SPLINE
SPL {X  -159.063, Y  +688.696, Z    +0.000, E1   -17.094, E3 +447767.075}
SPL {X  -159.987, Y  +672.488, Z    +0.000, E1    -5.638, E3 +447791.140}
SPL {X  -159.990, Y  +663.928, Z    +0.000, E1    +0.338, E3 +447796.935}
SPL {X  -159.990, Y  +658.009, Z    +0.000, E1    +4.774, E3 +447800.634}
SPL {X  -159.990, Y  +651.567, Z    +0.000, E1    +9.674, E3 +447806.038}
SPL {X  -159.990, Y  +638.711, Z    +0.000, E1   +17.883, E3 +447821.684}
SPL {X  -159.990, Y  +631.642, Z    +0.000, E1   +20.884, E3 +447837.242}
SPL {X  -159.990, Y  +626.048, Z    +0.000, E1   +22.026, E3 +447857.236}
SPL {X  -159.990, Y  +623.760, Z    +0.000, E1   +22.031, E3 +447869.223}
SPL {X  -159.990, Y  +621.334, Z    +0.000, E1   +22.029, E3 +447881.949}
SPL {X  -159.990, Y  +618.387, Z    +0.000, E1   +22.057, E3 +447897.339}
SPL {X  -159.990, Y  +615.830, Z    +0.000, E1   +22.023, E3 +447910.830}
SPL {X  -159.990, Y  +613.034, Z    +0.000, E1   +22.053, E3 +447925.437}
SPL {X  -159.990, Y  +609.503, Z    +0.000, E1   +22.054, E3 +447943.964}
SPL {X  -159.990, Y  +605.804, Z    +0.000, E1   +22.064, E3 +447963.308}
SPL {X  -159.990, Y  +602.819, Z    +0.000, E1   +22.037, E3 +447978.979}
SPL {X  -159.990, Y  +600.642, Z    +0.000, E1   +22.032, E3 +447990.407}
SPL {X  -159.990, Y  +598.568, Z    +0.000, E1   +22.046, E3 +448001.200}
SPL {X  -159.990, Y  +596.440, Z    +0.000, E1   +22.036, E3 +448012.381}
SPL {X  -159.990, Y  +593.768, Z    +0.000, E1   +22.071, E3 +448026.314}
SPL {X  -159.990, Y  +590.068, Z    +0.000, E1   +22.076, E3 +448045.683}
SPL {X  -159.990, Y  +587.130, Z    +0.000, E1   +22.046, E3 +448061.120}
SPL {X  -159.990, Y  +585.120, Z    +0.000, E1   +22.045, E3 +448071.621}
SPL {X  -159.990, Y  +583.118, Z    +0.000, E1   +22.052, E3 +448082.108}
SPL {X  -159.990, Y  +580.862, Z    +0.000, E1   +22.049, E3 +448093.946}
SPL {X  -159.990, Y  +578.386, Z    +0.000, E1   +22.057, E3 +448106.901}
SPL {X  -159.990, Y  +576.252, Z    +0.000, E1   +22.038, E3 +448118.124}
SPL {X  -159.990, Y  +574.280, Z    +0.000, E1   +22.051, E3 +448128.418}
SPL {X  -159.990, Y  +571.711, Z    +0.000, E1   +22.058, E3 +448141.892}
SPL {X  -159.990, Y  +569.285, Z    +0.000, E1   +22.044, E3 +448154.617}
SPL {X  -159.990, Y  +567.211, Z    +0.000, E1   +22.046, E3 +448165.478}
SPL {X  -159.990, Y  +565.039, Z    +0.000, E1   +22.047, E3 +448176.856}
SPL {X  -159.990, Y  +562.755, Z    +0.000, E1   +22.047, E3 +448188.841}
SPL {X  -159.990, Y  +560.652, Z    +0.000, E1   +22.038, E3 +448199.886}
SPL {X  -159.990, Y  +558.852, Z    +0.000, E1   +22.046, E3 +448209.258}
SPL {X  -159.990, Y  +556.672, Z    +0.000, E1   +22.055, E3 +448220.647}
SPL {X  -159.990, Y  +553.726, Z    +0.000, E1   +22.080, E3 +448236.010}
SPL {X  -159.990, Y  +550.886, Z    +0.000, E1   +22.056, E3 +448250.948}
SPL {X  -159.990, Y  +548.814, Z    +0.000, E1   +22.049, E3 +448261.794}
SPL {X  -159.990, Y  +546.122, Z    +0.000, E1   +22.088, E3 +448275.808}
SPL {X  -159.990, Y  +542.390, Z    +0.000, E1   +22.086, E3 +448295.390}
SPL {X  -159.990, Y  +539.341, Z    +0.000, E1   +22.056, E3 +448311.411}
SPL {X  -159.990, Y  +536.301, Z    +0.000, E1   +22.084, E3 +448327.266}
SPL {X  -159.990, Y  +533.389, Z    +0.000, E1   +22.057, E3 +448342.573}
SPL {X  -159.990, Y  +531.347, Z    +0.000, E1   +22.052, E3 +448353.274}
SPL {X  -159.990, Y  +529.626, Z    +0.000, E1   +22.051, E3 +448362.271}
SPL {X  -159.990, Y  +527.412, Z    +0.000, E1   +22.067, E3 +448373.824}
SPL {X  -159.990, Y  +524.425, Z    +0.000, E1   +22.078, E3 +448389.456}
SPL {X  -159.990, Y  +521.599, Z    +0.000, E1   +22.060, E3 +448404.298}
SPL {X  -159.990, Y  +519.209, Z    +0.000, E1   +22.063, E3 +448416.773}
SPL {X  -159.990, Y  +517.330, Z    +0.000, E1   +22.053, E3 +448426.629}
SPL {X  -159.990, Y  +514.729, Z    +0.000, E1   +22.089, E3 +448440.187}
SPL {X  -159.990, Y  +511.670, Z    +0.000, E1   +22.064, E3 +448456.274}
SPL {X  -159.990, Y  +506.947, Z    +0.000, E1   +23.726, E3 +448466.303}
SPL {X  -159.990, Y  +496.921, Z    +0.000, E1   +28.340, E3 +448475.052}
SPL {X  -159.990, Y  +495.822, Z    +0.000, E1   +27.449, E3 +448485.800}
SPL {X  -159.990, Y  +494.952, Z    +0.000, E1   +26.628, E3 +448495.383}
SPL {X  -159.990, Y  +493.896, Z    +0.000, E1   +25.736, E3 +448506.713}
SPL {X  -159.990, Y  +491.647, Z    +0.000, E1   +25.401, E3 +448519.248}
SPL {X  -159.990, Y  +488.807, Z    +0.000, E1   +25.397, E3 +448531.947}
SPL {X  -159.990, Y  +486.070, Z    +0.000, E1   +25.399, E3 +448544.177}
SPL {X  -159.990, Y  +482.821, Z    +0.000, E1   +25.411, E3 +448558.679}
SPL {X  -159.990, Y  +480.183, Z    +0.000, E1   +25.384, E3 +448570.519}
SPL {X  -159.990, Y  +477.508, Z    +0.000, E1   +25.410, E3 +448582.428}
SPL {X  -159.990, Y  +473.634, Z    +0.000, E1   +25.426, E3 +448599.717}
SPL {X  -159.990, Y  +470.047, Z    +0.000, E1   +25.402, E3 +448615.798}
SPL {X  -159.990, Y  +466.213, Z    +0.000, E1   +25.433, E3 +448632.878}
SPL {X  -159.990, Y  +462.520, Z    +0.000, E1   +25.400, E3 +448649.446}
SPL {X  -159.990, Y  +460.081, Z    +0.000, E1   +25.390, E3 +448660.348}
SPL {X  -159.990, Y  +457.497, Z    +0.000, E1   +25.403, E3 +448671.872}
SPL {X  -159.990, Y  +455.126, Z    +0.000, E1   +25.389, E3 +448682.481}
SPL {X  -159.990, Y  +452.123, Z    +0.000, E1   +25.426, E3 +448695.838}
SPL {X  -159.990, Y  +448.503, Z    +0.000, E1   +25.410, E3 +448712.040}
SPL {X  -159.990, Y  +445.882, Z    +0.000, E1   +25.385, E3 +448723.842}
SPL {X  -159.990, Y  +443.345, Z    +0.000, E1   +25.390, E3 +448735.224}
SPL {X  -159.990, Y  +440.220, Z    +0.000, E1   +25.392, E3 +448749.212}
SPL {X  -159.990, Y  +436.316, Z    +0.000, E1   +25.420, E3 +448766.616}
SPL {X  -159.990, Y  +432.613, Z    +0.000, E1   +25.390, E3 +448783.241}
SPL {X  -159.990, Y  +429.079, Z    +0.000, E1   +25.407, E3 +448799.012}
SPL {X  -159.990, Y  +425.142, Z    +0.000, E1   +25.407, E3 +448816.614}
SPL {X  -159.990, Y  +421.010, Z    +0.000, E1   +25.418, E3 +448835.075}
SPL {X  -159.990, Y  +417.514, Z    +0.000, E1   +25.386, E3 +448850.768}
SPL {X  -159.990, Y  +414.805, Z    +0.000, E1   +25.385, E3 +448862.888}
SPL {X  -159.990, Y  +411.959, Z    +0.000, E1   +25.386, E3 +448875.615}
SPL {X  -159.990, Y  +408.981, Z    +0.000, E1   +25.392, E3 +448888.919}
SPL {X  -159.990, Y  +406.574, Z    +0.000, E1   +25.375, E3 +448899.693}
SPL {X  -159.990, Y  +403.513, Z    +0.000, E1   +25.420, E3 +448913.292}
SPL {X  -159.990, Y  +399.257, Z    +0.000, E1   +25.420, E3 +448932.333}
SPL {X  -159.990, Y  +395.992, Z    +0.000, E1   +25.380, E3 +448947.022}
SPL {X  -159.990, Y  +393.569, Z    +0.000, E1   +25.379, E3 +448957.866}
SPL {X  -159.990, Y  +390.564, Z    +0.000, E1   +25.393, E3 +448971.310}
SPL {X  -159.990, Y  +387.503, Z    +0.000, E1   +25.378, E3 +448985.024}
SPL {X  -159.990, Y  +384.900, Z    +0.000, E1   +25.383, E3 +448996.634}
SPL {X  -159.990, Y  +382.110, Z    +0.000, E1   +25.393, E3 +449009.080}
SPL {X  -159.961, Y  +379.439, Z    +0.000, E1   +25.380, E3 +449021.060}
SPL {X  -159.894, Y  +376.959, Z    +0.000, E1   +25.370, E3 +449032.237}
SPL {X  -159.784, Y  +374.382, Z    +0.000, E1   +25.356, E3 +449043.878}
SPL {X  -159.621, Y  +371.640, Z    +0.000, E1   +25.335, E3 +449056.318}
SPL {X  -159.406, Y  +368.844, Z    +0.000, E1   +25.307, E3 +449069.031}
SPL {X  -159.144, Y  +366.072, Z    +0.000, E1   +25.281, E3 +449081.638}
SPL {X  -158.822, Y  +363.200, Z    +0.000, E1   +25.236, E3 +449094.811}
SPL {X  -158.491, Y  +360.654, Z    +0.000, E1   +25.188, E3 +449106.551}
SPL {X  -158.127, Y  +358.155, Z    +0.000, E1   +25.126, E3 +449118.171}
SPL {X  -158.095, Y  +357.947, Z    +0.000, E1   +21.741, E3 +449149.743}
ENDSPLINE

SPLINE
SPL {X  -158.454, Y  +360.384, Z    +0.000, E1   +19.366, E3 +449161.894}
SPL {X  -159.737, Y  +373.507, Z    +0.000, E1   +10.311, E3 +449183.929}
SPL {X  -159.990, Y  +382.574, Z    +0.000, E1    +4.463, E3 +449190.617}
SPL {X  -159.990, Y  +389.909, Z    +0.000, E1    -0.662, E3 +449194.632}
SPL {X  -159.990, Y  +396.289, Z    +0.000, E1    -5.500, E3 +449198.412}
SPL {X  -159.990, Y  +407.941, Z    +0.000, E1   -14.126, E3 +449209.749}
SPL {X  -159.990, Y  +418.671, Z    +0.000, E1   -19.855, E3 +449229.165}
SPL {X  -159.990, Y  +429.878, Z    +0.000, E1   -23.330, E3 +449259.220}
SPL {X  -159.990, Y  +432.766, Z    +0.000, E1   -23.321, E3 +449273.443}
SPL {X  -159.990, Y  +434.794, Z    +0.000, E1   -23.304, E3 +449283.474}
SPL {X  -159.990, Y  +437.007, Z    +0.000, E1   -23.323, E3 +449294.326}
SPL {X  -159.990, Y  +439.778, Z    +0.000, E1   -23.323, E3 +449307.959}
SPL {X  -159.990, Y  +442.010, Z    +0.000, E1   -23.308, E3 +449318.980}
SPL {X  -159.990, Y  +443.729, Z    +0.000, E1   -23.310, E3 +449327.436}
SPL {X  -159.990, Y  +446.037, Z    +0.000, E1   -23.324, E3 +449338.773}
SPL {X  -159.990, Y  +449.434, Z    +0.000, E1   -23.356, E3 +449355.394}
SPL {X  -159.990, Y  +453.256, Z    +0.000, E1   -23.349, E3 +449374.229}
SPL {X  -159.990, Y  +455.953, Z    +0.000, E1   -23.320, E3 +449387.543}
SPL {X  -159.990, Y  +458.265, Z    +0.000, E1   -23.328, E3 +449398.898}
SPL {X  -159.990, Y  +461.258, Z    +0.000, E1   -23.344, E3 +449413.614}
SPL {X  -159.990, Y  +464.382, Z    +0.000, E1   -23.332, E3 +449428.995}
SPL {X  -159.990, Y  +466.881, Z    +0.000, E1   -23.322, E3 +449441.315}
SPL {X  -159.990, Y  +468.951, Z    +0.000, E1   -23.319, E3 +449451.507}
SPL {X  -159.990, Y  +471.818, Z    +0.000, E1   -23.351, E3 +449465.554}
SPL {X  -159.990, Y  +474.801, Z    +0.000, E1   -23.320, E3 +449480.330}
SPL {X  -159.990, Y  +476.830, Z    +0.000, E1   -23.323, E3 +449490.309}
SPL {X  -159.990, Y  +479.553, Z    +0.000, E1   -23.328, E3 +449503.711}
SPL {X  -159.990, Y  +482.950, Z    +0.000, E1   -23.350, E3 +449520.383}
SPL {X  -159.990, Y  +486.109, Z    +0.000, E1   -23.322, E3 +449535.999}
SPL {X  -159.990, Y  +489.247, Z    +0.000, E1   -23.348, E3 +449551.386}
SPL {X  -159.990, Y  +493.031, Z    +0.000, E1   -23.350, E3 +449570.010}
SPL {X  -159.990, Y  +496.869, Z    +0.000, E1   -23.349, E3 +449588.900}
SPL {X  -159.990, Y  +499.995, Z    +0.000, E1   -23.324, E3 +449604.334}
SPL {X  -159.990, Y  +502.456, Z    +0.000, E1   -23.324, E3 +449616.448}
SPL {X  -159.990, Y  +505.646, Z    +0.000, E1   -23.350, E3 +449632.103}
SPL {X  -159.990, Y  +508.862, Z    +0.000, E1   -23.328, E3 +449647.968}
SPL {X  -159.990, Y  +511.771, Z    +0.000, E1   -23.331, E3 +449662.290}
SPL {X  -159.990, Y  +514.016, Z    +0.000, E1   -23.308, E3 +449673.394}
SPL {X  -159.990, Y  +516.860, Z    +0.000, E1   -23.355, E3 +449687.280}
SPL {X  -159.990, Y  +520.719, Z    +0.000, E1   -23.363, E3 +449706.190}
SPL {X  -159.990, Y  +523.968, Z    +0.000, E1   -23.332, E3 +449722.275}
SPL {X  -159.990, Y  +526.466, Z    +0.000, E1   -23.320, E3 +449734.618}
SPL {X  -159.990, Y  +528.815, Z    +0.000, E1   -23.322, E3 +449746.178}
SPL {X  -159.990, Y  +531.246, Z    +0.000, E1   -23.325, E3 +449758.116}
SPL {X  -159.990, Y  +534.143, Z    +0.000, E1   -23.341, E3 +449772.351}
SPL {X  -159.990, Y  +537.024, Z    +0.000, E1   -23.321, E3 +449786.595}
SPL {X  -159.990, Y  +539.129, Z    +0.000, E1   -23.310, E3 +449796.978}
SPL {X  -159.990, Y  +541.882, Z    +0.000, E1   -23.346, E3 +449810.459}
SPL {X  -159.990, Y  +544.941, Z    +0.000, E1   -23.325, E3 +449825.541}
SPL {X  -159.990, Y  +548.126, Z    +0.000, E1   -23.354, E3 +449841.158}
SPL {X  -159.990, Y  +551.344, Z    +0.000, E1   -23.327, E3 +449857.050}
SPL {X  -159.990, Y  +553.642, Z    +0.000, E1   -23.319, E3 +449868.368}
SPL {X  -159.990, Y  +556.481, Z    +0.000, E1   -23.354, E3 +449882.275}
SPL {X  -159.990, Y  +559.475, Z    +0.000, E1   -23.321, E3 +449897.081}
SPL {X  -159.990, Y  +561.830, Z    +0.000, E1   -23.325, E3 +449908.666}
SPL {X  -159.990, Y  +564.273, Z    +0.000, E1   -23.325, E3 +449920.690}
SPL {X  -159.990, Y  +566.342, Z    +0.000, E1   -23.314, E3 +449930.894}
SPL {X  -159.990, Y  +568.849, Z    +0.000, E1   -23.338, E3 +449943.189}
SPL {X  -159.990, Y  +572.204, Z    +0.000, E1   -23.344, E3 +449959.684}
SPL {X  -159.990, Y  +575.097, Z    +0.000, E1   -23.325, E3 +449973.961}
SPL {X  -159.990, Y  +578.356, Z    +0.000, E1   -23.358, E3 +449989.933}
SPL {X  -159.990, Y  +582.292, Z    +0.000, E1   -23.360, E3 +450009.249}
SPL {X  -159.990, Y  +585.165, Z    +0.000, E1   -23.322, E3 +450023.492}
SPL {X  -159.990, Y  +587.388, Z    +0.000, E1   -23.328, E3 +450034.405}
SPL {X  -159.990, Y  +590.594, Z    +0.000, E1   -23.363, E3 +450050.097}
SPL {X  -159.990, Y  +594.301, Z    +0.000, E1   -23.358, E3 +450068.302}
SPL {X  -159.990, Y  +597.981, Z    +0.000, E1   -23.373, E3 +450086.350}
SPL {X  -159.990, Y  +600.935, Z    +0.000, E1   -23.343, E3 +450100.882}
SPL {X  -159.990, Y  +603.047, Z    +0.000, E1   -23.344, E3 +450111.268}
SPL {X  -159.990, Y  +605.187, Z    +0.000, E1   -23.344, E3 +450121.790}
SPL {X  -159.990, Y  +607.319, Z    +0.000, E1   -23.353, E3 +450132.252}
SPL {X  -159.990, Y  +610.569, Z    +0.000, E1   -23.372, E3 +450148.217}
SPL {X  -159.990, Y  +613.591, Z    +0.000, E1   -23.342, E3 +450163.145}
SPL {X  -159.990, Y  +615.604, Z    +0.000, E1   -23.330, E3 +450173.083}
SPL {X  -159.990, Y  +617.623, Z    +0.000, E1   -23.337, E3 +450183.014}
SPL {X  -159.990, Y  +620.788, Z    +0.000, E1   -23.368, E3 +450198.519}
SPL {X  -159.990, Y  +623.764, Z    +0.000, E1   -23.335, E3 +450213.211}
SPL {X  -159.990, Y  +626.608, Z    +0.000, E1   -23.361, E3 +450227.136}
SPL {X  -159.990, Y  +630.271, Z    +0.000, E1   -23.375, E3 +450245.097}
SPL {X  -159.990, Y  +633.318, Z    +0.000, E1   -23.339, E3 +450260.175}
SPL {X  -159.990, Y  +635.650, Z    +0.000, E1   -23.339, E3 +450271.646}
SPL {X  -159.990, Y  +637.839, Z    +0.000, E1   -23.335, E3 +450282.456}
SPL {X  -159.990, Y  +640.072, Z    +0.000, E1   -23.325, E3 +450293.488}
SPL {X  -159.990, Y  +642.230, Z    +0.000, E1   -23.323, E3 +450304.170}
SPL {X  -159.990, Y  +645.287, Z    +0.000, E1   -23.340, E3 +450319.196}
SPL {X  -159.990, Y  +648.792, Z    +0.000, E1   -23.346, E3 +450336.454}
SPL {X  -159.990, Y  +652.623, Z    +0.000, E1   -23.348, E3 +450355.289}
SPL {X  -159.990, Y  +656.380, Z    +0.000, E1   -23.347, E3 +450373.784}
SPL {X  -159.990, Y  +659.180, Z    +0.000, E1   -23.314, E3 +450387.632}
SPL {X  -159.990, Y  +661.392, Z    +0.000, E1   -23.318, E3 +450398.526}
SPL {X  -159.990, Y  +663.662, Z    +0.000, E1   -23.322, E3 +450409.650}
SPL {X  -159.990, Y  +665.964, Z    +0.000, E1   -23.328, E3 +450420.940}
SPL {X  -159.990, Y  +668.989, Z    +0.000, E1   -23.359, E3 +450435.776}
SPL {X  -159.990, Y  +671.893, Z    +0.000, E1   -23.319, E3 +450450.156}
SPL {X  -159.974, Y  +673.789, Z    +0.000, E1   -23.323, E3 +450459.472}
SPL {X  -159.924, Y  +676.110, Z    +0.000, E1   -23.320, E3 +450470.957}
SPL {X  -159.801, Y  +679.265, Z    +0.000, E1   -23.327, E3 +450486.575}
SPL {X  -159.626, Y  +682.287, Z    +0.000, E1   -23.280, E3 +450501.674}
SPL {X  -159.462, Y  +684.486, Z    +0.000, E1   -23.258, E3 +450512.673}
SPL {X  -159.246, Y  +686.911, Z    +0.000, E1   -23.230, E3 +450524.835}
SPL {X  -159.019, Y  +689.098, Z    +0.000, E1   -23.200, E3 +450535.837}
SPL {X  -158.660, Y  +692.086, Z    +0.000, E1   -23.176, E3 +450550.881}
ENDSPLINE

SPLINE
SPL {X  -159.063, Y  +688.696, Z    +0.000, E1   -17.094, E3 +450593.162}
SPL {X  -159.967, Y  +674.206, Z    +0.000, E1    -6.731, E3 +450615.975}
SPL {X  -159.990, Y  +665.270, Z    +0.000, E1    -0.699, E3 +450622.144}
SPL {X  -159.990, Y  +658.009, Z    +0.000, E1    +4.774, E3 +450626.721}
SPL {X  -159.990, Y  +651.567, Z    +0.000, E1    +9.674, E3 +450632.125}
SPL {X  -159.990, Y  +637.762, Z    +0.000, E1   +18.345, E3 +450649.483}
SPL {X  -159.990, Y  +626.382, Z    +0.000, E1   +22.040, E3 +450681.532}
SPL {X  -159.990, Y  +623.760, Z    +0.000, E1   +22.031, E3 +450695.310}
SPL {X  -159.990, Y  +621.334, Z    +0.000, E1   +22.029, E3 +450708.036}
SPL {X  -159.990, Y  +618.387, Z    +0.000, E1   +22.057, E3 +450723.426}
SPL {X  -159.990, Y  +614.928, Z    +0.000, E1   +22.055, E3 +450741.579}
SPL {X  -159.990, Y  +611.459, Z    +0.000, E1   +22.053, E3 +450759.782}
SPL {X  -159.990, Y  +608.810, Z    +0.000, E1   +22.023, E3 +450773.750}
SPL {X  -159.990, Y  +606.481, Z    +0.000, E1   +22.033, E3 +450785.925}
SPL {X  -159.990, Y  +603.419, Z    +0.000, E1   +22.064, E3 +450801.865}
SPL {X  -159.990, Y  +600.642, Z    +0.000, E1   +22.032, E3 +450816.494}
SPL {X  -159.990, Y  +598.568, Z    +0.000, E1   +22.046, E3 +450827.287}
SPL {X  -159.990, Y  +595.493, Z    +0.000, E1   +22.070, E3 +450843.370}
SPL {X  -159.990, Y  +592.865, Z    +0.000, E1   +22.036, E3 +450857.199}
SPL {X  -159.990, Y  +590.803, Z    +0.000, E1   +22.046, E3 +450867.989}
SPL {X  -159.990, Y  +587.778, Z    +0.000, E1   +22.073, E3 +450883.764}
SPL {X  -159.990, Y  +585.120, Z    +0.000, E1   +22.045, E3 +450897.708}
SPL {X  -159.990, Y  +583.118, Z    +0.000, E1   +22.052, E3 +450908.195}
SPL {X  -159.990, Y  +580.131, Z    +0.000, E1   +22.078, E3 +450923.801}
SPL {X  -159.990, Y  +576.888, Z    +0.000, E1   +22.061, E3 +450940.831}
SPL {X  -159.990, Y  +574.280, Z    +0.000, E1   +22.051, E3 +450954.505}
SPL {X  -159.990, Y  +571.711, Z    +0.000, E1   +22.058, E3 +450967.979}
SPL {X  -159.990, Y  +569.285, Z    +0.000, E1   +22.044, E3 +450980.704}
SPL {X  -159.990, Y  +567.211, Z    +0.000, E1   +22.046, E3 +450991.565}
SPL {X  -159.990, Y  +565.039, Z    +0.000, E1   +22.047, E3 +451002.942}
SPL {X  -159.990, Y  +562.755, Z    +0.000, E1   +22.047, E3 +451014.928}
SPL {X  -159.990, Y  +560.652, Z    +0.000, E1   +22.038, E3 +451025.973}
SPL {X  -159.990, Y  +558.852, Z    +0.000, E1   +22.046, E3 +451035.345}
SPL {X  -159.990, Y  +556.672, Z    +0.000, E1   +22.055, E3 +451046.734}
SPL {X  -159.990, Y  +553.726, Z    +0.000, E1   +22.080, E3 +451062.097}
SPL {X  -159.990, Y  +550.886, Z    +0.000, E1   +22.056, E3 +451077.035}
SPL {X  -159.990, Y  +548.814, Z    +0.000, E1   +22.049, E3 +451087.881}
SPL {X  -159.990, Y  +546.122, Z    +0.000, E1   +22.088, E3 +451101.895}
SPL {X  -159.990, Y  +542.390, Z    +0.000, E1   +22.086, E3 +451121.477}
SPL {X  -159.990, Y  +539.341, Z    +0.000, E1   +22.056, E3 +451137.498}
SPL {X  -159.990, Y  +536.984, Z    +0.000, E1   +22.057, E3 +451149.829}
SPL {X  -159.990, Y  +534.045, Z    +0.000, E1   +22.087, E3 +451165.154}
SPL {X  -159.990, Y  +530.476, Z    +0.000, E1   +22.084, E3 +451183.847}
SPL {X  -159.990, Y  +527.412, Z    +0.000, E1   +22.067, E3 +451199.911}
SPL {X  -159.990, Y  +524.425, Z    +0.000, E1   +22.078, E3 +451215.543}
SPL {X  -159.990, Y  +521.599, Z    +0.000, E1   +22.060, E3 +451230.385}
SPL {X  -159.990, Y  +519.209, Z    +0.000, E1   +22.063, E3 +451242.860}
SPL {X  -159.990, Y  +516.651, Z    +0.000, E1   +22.071, E3 +451256.239}
SPL {X  -159.990, Y  +514.122, Z    +0.000, E1   +22.061, E3 +451269.512}
SPL {X  -159.990, Y  +511.670, Z    +0.000, E1   +22.064, E3 +451282.361}
SPL {X  -159.990, Y  +506.947, Z    +0.000, E1   +23.726, E3 +451292.390}
SPL {X  -159.990, Y  +496.921, Z    +0.000, E1   +28.340, E3 +451301.139}
SPL {X  -159.990, Y  +495.822, Z    +0.000, E1   +27.449, E3 +451311.887}
SPL {X  -159.990, Y  +494.952, Z    +0.000, E1   +26.628, E3 +451321.470}
SPL {X  -159.990, Y  +493.896, Z    +0.000, E1   +25.736, E3 +451332.800}
SPL {X  -159.990, Y  +491.647, Z    +0.000, E1   +25.401, E3 +451345.335}
SPL {X  -159.990, Y  +488.807, Z    +0.000, E1   +25.397, E3 +451358.033}
SPL {X  -159.990, Y  +486.070, Z    +0.000, E1   +25.399, E3 +451370.264}
SPL {X  -159.990, Y  +483.747, Z    +0.000, E1   +25.384, E3 +451380.677}
SPL {X  -159.990, Y  +481.038, Z    +0.000, E1   +25.412, E3 +451392.733}
SPL {X  -159.990, Y  +477.508, Z    +0.000, E1   +25.410, E3 +451408.515}
SPL {X  -159.990, Y  +473.634, Z    +0.000, E1   +25.426, E3 +451425.804}
SPL {X  -159.990, Y  +470.047, Z    +0.000, E1   +25.402, E3 +451441.885}
SPL {X  -159.990, Y  +467.082, Z    +0.000, E1   +25.399, E3 +451455.132}
SPL {X  -159.990, Y  +464.063, Z    +0.000, E1   +25.405, E3 +451468.627}
SPL {X  -159.990, Y  +460.712, Z    +0.000, E1   +25.411, E3 +451483.587}
SPL {X  -159.990, Y  +457.497, Z    +0.000, E1   +25.403, E3 +451497.959}
SPL {X  -159.990, Y  +454.323, Z    +0.000, E1   +25.412, E3 +451512.118}
SPL {X  -159.990, Y  +450.823, Z    +0.000, E1   +25.417, E3 +451527.747}
SPL {X  -159.990, Y  +447.982, Z    +0.000, E1   +25.393, E3 +451540.488}
SPL {X  -159.990, Y  +445.108, Z    +0.000, E1   +25.407, E3 +451553.365}
SPL {X  -159.990, Y  +441.797, Z    +0.000, E1   +25.390, E3 +451568.244}
SPL {X  -159.990, Y  +439.442, Z    +0.000, E1   +25.369, E3 +451578.821}
SPL {X  -159.990, Y  +436.316, Z    +0.000, E1   +25.420, E3 +451592.703}
SPL {X  -159.990, Y  +432.613, Z    +0.000, E1   +25.390, E3 +451609.328}
SPL {X  -159.990, Y  +429.827, Z    +0.000, E1   +25.380, E3 +451621.805}
SPL {X  -159.990, Y  +426.865, Z    +0.000, E1   +25.398, E3 +451635.010}
SPL {X  -159.990, Y  +423.417, Z    +0.000, E1   +25.400, E3 +451650.426}
SPL {X  -159.990, Y  +420.283, Z    +0.000, E1   +25.386, E3 +451664.470}
SPL {X  -159.990, Y  +417.514, Z    +0.000, E1   +25.386, E3 +451676.855}
SPL {X  -159.990, Y  +414.805, Z    +0.000, E1   +25.385, E3 +451688.975}
SPL {X  -159.990, Y  +411.959, Z    +0.000, E1   +25.386, E3 +451701.702}
SPL {X  -159.990, Y  +408.981, Z    +0.000, E1   +25.392, E3 +451715.006}
SPL {X  -159.990, Y  +405.773, Z    +0.000, E1   +25.398, E3 +451729.315}
SPL {X  -159.990, Y  +402.805, Z    +0.000, E1   +25.389, E3 +451742.602}
SPL {X  -159.990, Y  +399.257, Z    +0.000, E1   +25.420, E3 +451758.420}
SPL {X  -159.990, Y  +395.992, Z    +0.000, E1   +25.380, E3 +451773.109}
SPL {X  -159.990, Y  +393.569, Z    +0.000, E1   +25.379, E3 +451783.952}
SPL {X  -159.990, Y  +390.564, Z    +0.000, E1   +25.393, E3 +451797.397}
SPL {X  -159.990, Y  +387.503, Z    +0.000, E1   +25.378, E3 +451811.111}
SPL {X  -159.990, Y  +384.900, Z    +0.000, E1   +25.383, E3 +451822.721}
SPL {X  -159.990, Y  +382.110, Z    +0.000, E1   +25.393, E3 +451835.167}
SPL {X  -159.961, Y  +379.439, Z    +0.000, E1   +25.380, E3 +451847.147}
SPL {X  -159.894, Y  +376.959, Z    +0.000, E1   +25.370, E3 +451858.324}
SPL {X  -159.784, Y  +374.382, Z    +0.000, E1   +25.356, E3 +451869.965}
SPL {X  -159.621, Y  +371.640, Z    +0.000, E1   +25.335, E3 +451882.405}
SPL {X  -159.406, Y  +368.844, Z    +0.000, E1   +25.307, E3 +451895.118}
SPL {X  -159.144, Y  +366.072, Z    +0.000, E1   +25.281, E3 +451907.725}
SPL {X  -158.822, Y  +363.200, Z    +0.000, E1   +25.236, E3 +451920.898}
SPL {X  -158.491, Y  +360.654, Z    +0.000, E1   +25.188, E3 +451932.638}
SPL {X  -158.127, Y  +358.155, Z    +0.000, E1   +25.126, E3 +451944.258}
SPL {X  -158.095, Y  +357.947, Z    +0.000, E1   +21.741, E3 +451975.830}
ENDSPLINE

SPLINE
SPL {X  -158.454, Y  +360.384, Z    +0.000, E1   +19.366, E3 +451987.981}
SPL {X  -159.737, Y  +373.507, Z    +0.000, E1   +10.311, E3 +452010.016}
SPL {X  -159.990, Y  +382.574, Z    +0.000, E1    +4.463, E3 +452016.704}
SPL {X  -159.990, Y  +387.496, Z    +0.000, E1    +1.004, E3 +452019.449}
SPL {X  -159.990, Y  +395.121, Z    +0.000, E1    -4.514, E3 +452023.761}
SPL {X  -159.990, Y  +407.941, Z    +0.000, E1   -14.126, E3 +452035.836}
SPL {X  -159.990, Y  +418.671, Z    +0.000, E1   -19.855, E3 +452055.252}
SPL {X  -159.990, Y  +428.534, Z    +0.000, E1   -23.299, E3 +452078.772}
SPL {X  -159.990, Y  +430.313, Z    +0.000, E1   -23.313, E3 +452087.485}
SPL {X  -159.990, Y  +432.766, Z    +0.000, E1   -23.321, E3 +452099.530}
SPL {X  -159.990, Y  +434.794, Z    +0.000, E1   -23.304, E3 +452109.561}
SPL {X  -159.990, Y  +437.007, Z    +0.000, E1   -23.323, E3 +452120.413}
SPL {X  -159.990, Y  +439.778, Z    +0.000, E1   -23.323, E3 +452134.046}
SPL {X  -159.990, Y  +442.010, Z    +0.000, E1   -23.308, E3 +452145.067}
SPL {X  -159.990, Y  +443.729, Z    +0.000, E1   -23.310, E3 +452153.523}
SPL {X  -159.990, Y  +446.037, Z    +0.000, E1   -23.324, E3 +452164.860}
SPL {X  -159.990, Y  +449.434, Z    +0.000, E1   -23.356, E3 +452181.481}
SPL {X  -159.990, Y  +453.256, Z    +0.000, E1   -23.349, E3 +452200.316}
SPL {X  -159.990, Y  +455.953, Z    +0.000, E1   -23.320, E3 +452213.630}
SPL {X  -159.990, Y  +458.265, Z    +0.000, E1   -23.328, E3 +452224.985}
SPL {X  -159.990, Y  +461.258, Z    +0.000, E1   -23.344, E3 +452239.701}
SPL {X  -159.990, Y  +464.382, Z    +0.000, E1   -23.332, E3 +452255.082}
SPL {X  -159.990, Y  +466.881, Z    +0.000, E1   -23.322, E3 +452267.402}
SPL {X  -159.990, Y  +468.951, Z    +0.000, E1   -23.319, E3 +452277.594}
SPL {X  -159.990, Y  +470.991, Z    +0.000, E1   -23.322, E3 +452287.624}
SPL {X  -159.990, Y  +474.027, Z    +0.000, E1   -23.352, E3 +452302.528}
SPL {X  -159.990, Y  +477.600, Z    +0.000, E1   -23.351, E3 +452320.131}
SPL {X  -159.990, Y  +481.169, Z    +0.000, E1   -23.337, E3 +452337.729}
SPL {X  -159.990, Y  +483.782, Z    +0.000, E1   -23.316, E3 +452350.633}
SPL {X  -159.990, Y  +486.109, Z    +0.000, E1   -23.322, E3 +452362.086}
SPL {X  -159.990, Y  +489.247, Z    +0.000, E1   -23.348, E3 +452377.473}
SPL {X  -159.990, Y  +493.031, Z    +0.000, E1   -23.350, E3 +452396.097}
SPL {X  -159.990, Y  +496.869, Z    +0.000, E1   -23.349, E3 +452414.987}
SPL {X  -159.990, Y  +499.995, Z    +0.000, E1   -23.324, E3 +452430.421}
SPL {X  -159.990, Y  +502.456, Z    +0.000, E1   -23.324, E3 +452442.535}
SPL {X  -159.990, Y  +505.646, Z    +0.000, E1   -23.350, E3 +452458.190}
SPL {X  -159.990, Y  +508.862, Z    +0.000, E1   -23.328, E3 +452474.055}
SPL {X  -159.990, Y  +511.771, Z    +0.000, E1   -23.331, E3 +452488.377}
SPL {X  -159.990, Y  +514.016, Z    +0.000, E1   -23.308, E3 +452499.481}
SPL {X  -159.990, Y  +516.860, Z    +0.000, E1   -23.355, E3 +452513.367}
SPL {X  -159.990, Y  +520.719, Z    +0.000, E1   -23.363, E3 +452532.277}
SPL {X  -159.990, Y  +523.968, Z    +0.000, E1   -23.332, E3 +452548.362}
SPL {X  -159.990, Y  +526.466, Z    +0.000, E1   -23.320, E3 +452560.705}
SPL {X  -159.990, Y  +528.815, Z    +0.000, E1   -23.322, E3 +452572.265}
SPL {X  -159.990, Y  +531.246, Z    +0.000, E1   -23.325, E3 +452584.203}
SPL {X  -159.990, Y  +533.354, Z    +0.000, E1   -23.318, E3 +452594.589}
SPL {X  -159.990, Y  +534.931, Z    +0.000, E1   -23.312, E3 +452602.383}
SPL {X  -159.990, Y  +537.024, Z    +0.000, E1   -23.321, E3 +452612.682}
SPL {X  -159.990, Y  +539.129, Z    +0.000, E1   -23.310, E3 +452623.065}
SPL {X  -159.990, Y  +541.183, Z    +0.000, E1   -23.319, E3 +452633.161}
SPL {X  -159.990, Y  +544.314, Z    +0.000, E1   -23.352, E3 +452648.490}
SPL {X  -159.990, Y  +548.126, Z    +0.000, E1   -23.354, E3 +452667.245}
SPL {X  -159.990, Y  +551.344, Z    +0.000, E1   -23.327, E3 +452683.137}
SPL {X  -159.990, Y  +553.642, Z    +0.000, E1   -23.319, E3 +452694.455}
SPL {X  -159.990, Y  +556.481, Z    +0.000, E1   -23.354, E3 +452708.362}
SPL {X  -159.990, Y  +559.475, Z    +0.000, E1   -23.321, E3 +452723.168}
SPL {X  -159.990, Y  +561.830, Z    +0.000, E1   -23.325, E3 +452734.752}
SPL {X  -159.990, Y  +564.273, Z    +0.000, E1   -23.325, E3 +452746.777}
SPL {X  -159.990, Y  +567.351, Z    +0.000, E1   -23.348, E3 +452761.873}
SPL {X  -159.990, Y  +570.560, Z    +0.000, E1   -23.333, E3 +452777.702}
SPL {X  -159.990, Y  +572.975, Z    +0.000, E1   -23.316, E3 +452789.621}
SPL {X  -159.990, Y  +575.097, Z    +0.000, E1   -23.325, E3 +452800.048}
SPL {X  -159.990, Y  +577.540, Z    +0.000, E1   -23.325, E3 +452812.077}
SPL {X  -159.990, Y  +580.312, Z    +0.000, E1   -23.340, E3 +452825.659}
SPL {X  -159.990, Y  +583.018, Z    +0.000, E1   -23.331, E3 +452838.964}
SPL {X  -159.990, Y  +585.165, Z    +0.000, E1   -23.322, E3 +452849.579}
SPL {X  -159.990, Y  +587.388, Z    +0.000, E1   -23.328, E3 +452860.492}
SPL {X  -159.990, Y  +589.763, Z    +0.000, E1   -23.328, E3 +452872.179}
SPL {X  -159.990, Y  +592.397, Z    +0.000, E1   -23.344, E3 +452885.060}
SPL {X  -159.990, Y  +595.589, Z    +0.000, E1   -23.356, E3 +452900.732}
SPL {X  -159.990, Y  +598.571, Z    +0.000, E1   -23.347, E3 +452915.376}
SPL {X  -159.990, Y  +600.935, Z    +0.000, E1   -23.343, E3 +452926.969}
SPL {X  -159.990, Y  +603.047, Z    +0.000, E1   -23.344, E3 +452937.355}
SPL {X  -159.990, Y  +605.187, Z    +0.000, E1   -23.344, E3 +452947.877}
SPL {X  -159.990, Y  +607.319, Z    +0.000, E1   -23.353, E3 +452958.339}
SPL {X  -159.990, Y  +609.514, Z    +0.000, E1   -23.337, E3 +452969.168}
SPL {X  -159.990, Y  +611.376, Z    +0.000, E1   -23.336, E3 +452978.355}
SPL {X  -159.990, Y  +613.591, Z    +0.000, E1   -23.342, E3 +452989.232}
SPL {X  -159.990, Y  +615.604, Z    +0.000, E1   -23.330, E3 +452999.170}
SPL {X  -159.990, Y  +617.623, Z    +0.000, E1   -23.337, E3 +453009.101}
SPL {X  -159.990, Y  +620.788, Z    +0.000, E1   -23.368, E3 +453024.606}
SPL {X  -159.990, Y  +623.764, Z    +0.000, E1   -23.335, E3 +453039.298}
SPL {X  -159.990, Y  +625.941, Z    +0.000, E1   -23.337, E3 +453049.990}
SPL {X  -159.990, Y  +628.611, Z    +0.000, E1   -23.357, E3 +453063.068}
SPL {X  -159.990, Y  +631.169, Z    +0.000, E1   -23.338, E3 +453075.673}
SPL {X  -159.990, Y  +633.318, Z    +0.000, E1   -23.339, E3 +453086.262}
SPL {X  -159.990, Y  +635.650, Z    +0.000, E1   -23.339, E3 +453097.733}
SPL {X  -159.990, Y  +637.839, Z    +0.000, E1   -23.335, E3 +453108.543}
SPL {X  -159.990, Y  +640.072, Z    +0.000, E1   -23.325, E3 +453119.575}
SPL {X  -159.990, Y  +642.230, Z    +0.000, E1   -23.323, E3 +453130.257}
SPL {X  -159.990, Y  +645.287, Z    +0.000, E1   -23.340, E3 +453145.282}
SPL {X  -159.990, Y  +648.792, Z    +0.000, E1   -23.346, E3 +453162.541}
SPL {X  -159.990, Y  +652.623, Z    +0.000, E1   -23.348, E3 +453181.376}
SPL {X  -159.990, Y  +656.380, Z    +0.000, E1   -23.347, E3 +453199.871}
SPL {X  -159.990, Y  +659.180, Z    +0.000, E1   -23.314, E3 +453213.719}
SPL {X  -159.990, Y  +661.392, Z    +0.000, E1   -23.318, E3 +453224.613}
SPL {X  -159.990, Y  +663.662, Z    +0.000, E1   -23.322, E3 +453235.737}
SPL {X  -159.990, Y  +665.964, Z    +0.000, E1   -23.328, E3 +453247.027}
SPL {X  -159.990, Y  +668.989, Z    +0.000, E1   -23.359, E3 +453261.863}
SPL {X  -159.983, Y  +672.946, Z    +0.000, E1   -23.359, E3 +453281.344}
SPL {X  -159.924, Y  +676.110, Z    +0.000, E1   -23.320, E3 +453297.044}
SPL {X  -159.801, Y  +679.265, Z    +0.000, E1   -23.327, E3 +453312.662}
SPL {X  -159.626, Y  +682.287, Z    +0.000, E1   -23.280, E3 +453327.761}
SPL {X  -159.462, Y  +684.486, Z    +0.000, E1   -23.258, E3 +453338.760}
SPL {X  -159.246, Y  +686.911, Z    +0.000, E1   -23.230, E3 +453350.922}
SPL {X  -159.019, Y  +689.098, Z    +0.000, E1   -23.200, E3 +453361.924}
SPL {X  -158.660, Y  +692.086, Z    +0.000, E1   -23.176, E3 +453376.968}
ENDSPLINE

SPLINE
SPL {X  -159.063, Y  +688.696, Z    +0.000, E1   -17.094, E3 +453419.249}
SPL {X  -159.967, Y  +674.206, Z    +0.000, E1    -6.731, E3 +453442.062}
SPL {X  -159.990, Y  +665.270, Z    +0.000, E1    -0.699, E3 +453448.231}
SPL {X  -159.990, Y  +658.009, Z    +0.000, E1    +4.774, E3 +453452.808}
SPL {X  -159.990, Y  +651.567, Z    +0.000, E1    +9.674, E3 +453458.212}
SPL {X  -159.990, Y  +637.762, Z    +0.000, E1   +18.345, E3 +453475.570}
SPL {X  -159.990, Y  +626.382, Z    +0.000, E1   +22.040, E3 +453507.619}
SPL {X  -159.990, Y  +623.760, Z    +0.000, E1   +22.031, E3 +453521.397}
SPL {X  -159.990, Y  +621.334, Z    +0.000, E1   +22.029, E3 +453534.123}
SPL {X  -159.990, Y  +619.505, Z    +0.000, E1   +22.018, E3 +453543.739}
SPL {X  -159.990, Y  +617.621, Z    +0.000, E1   +22.025, E3 +453553.604}
SPL {X  -159.990, Y  +614.928, Z    +0.000, E1   +22.055, E3 +453567.666}
SPL {X  -159.990, Y  +611.459, Z    +0.000, E1   +22.053, E3 +453585.869}
SPL {X  -159.990, Y  +608.810, Z    +0.000, E1   +22.023, E3 +453599.837}
SPL {X  -159.990, Y  +605.804, Z    +0.000, E1   +22.064, E3 +453615.482}
SPL {X  -159.990, Y  +602.819, Z    +0.000, E1   +22.037, E3 +453631.153}
SPL {X  -159.990, Y  +600.642, Z    +0.000, E1   +22.032, E3 +453642.581}
SPL {X  -159.990, Y  +598.568, Z    +0.000, E1   +22.046, E3 +453653.374}
SPL {X  -159.990, Y  +596.440, Z    +0.000, E1   +22.036, E3 +453664.555}
SPL {X  -159.990, Y  +593.768, Z    +0.000, E1   +22.071, E3 +453678.488}
SPL {X  -159.990, Y  +590.068, Z    +0.000, E1   +22.076, E3 +453697.857}
SPL {X  -159.990, Y  +587.130, Z    +0.000, E1   +22.046, E3 +453713.293}
SPL {X  -159.990, Y  +585.120, Z    +0.000, E1   +22.045, E3 +453723.795}
SPL {X  -159.990, Y  +583.118, Z    +0.000, E1   +22.052, E3 +453734.282}
SPL {X  -159.990, Y  +580.862, Z    +0.000, E1   +22.049, E3 +453746.119}
SPL {X  -159.990, Y  +578.386, Z    +0.000, E1   +22.057, E3 +453759.075}
SPL {X  -159.990, Y  +576.252, Z    +0.000, E1   +22.038, E3 +453770.298}
SPL {X  -159.990, Y  +574.280, Z    +0.000, E1   +22.051, E3 +453780.592}
SPL {X  -159.990, Y  +571.711, Z    +0.000, E1   +22.058, E3 +453794.066}
SPL {X  -159.990, Y  +569.285, Z    +0.000, E1   +22.044, E3 +453806.791}
SPL {X  -159.990, Y  +567.211, Z    +0.000, E1   +22.046, E3 +453817.652}
SPL {X  -159.990, Y  +565.039, Z    +0.000, E1   +22.047, E3 +453829.029}
SPL {X  -159.990, Y  +562.755, Z    +0.000, E1   +22.047, E3 +453841.015}
SPL {X  -159.990, Y  +560.652, Z    +0.000, E1   +22.038, E3 +453852.060}
SPL {X  -159.990, Y  +558.852, Z    +0.000, E1   +22.046, E3 +453861.432}
SPL {X  -159.990, Y  +556.672, Z    +0.000, E1   +22.055, E3 +453872.821}
SPL {X  -159.990, Y  +553.726, Z    +0.000, E1   +22.080, E3 +453888.184}
SPL {X  -159.990, Y  +550.886, Z    +0.000, E1   +22.056, E3 +453903.122}
SPL {X  -159.990, Y  +548.814, Z    +0.000, E1   +22.049, E3 +453913.968}
SPL {X  -159.990, Y  +546.122, Z    +0.000, E1   +22.088, E3 +453927.982}
SPL {X  -159.990, Y  +542.390, Z    +0.000, E1   +22.086, E3 +453947.564}
SPL {X  -159.990, Y  +539.341, Z    +0.000, E1   +22.056, E3 +453963.585}
SPL {X  -159.990, Y  +536.984, Z    +0.000, E1   +22.057, E3 +453975.916}
SPL {X  -159.990, Y  +534.045, Z    +0.000, E1   +22.087, E3 +453991.241}
SPL {X  -159.990, Y  +530.476, Z    +0.000, E1   +22.084, E3 +454009.934}
SPL {X  -159.990, Y  +527.412, Z    +0.000, E1   +22.067, E3 +454025.998}
SPL {X  -159.990, Y  +525.349, Z    +0.000, E1   +22.050, E3 +454036.839}
SPL {X  -159.990, Y  +523.717, Z    +0.000, E1   +22.050, E3 +454045.404}
SPL {X  -159.990, Y  +521.599, Z    +0.000, E1   +22.060, E3 +454056.472}
SPL {X  -159.990, Y  +519.209, Z    +0.000, E1   +22.063, E3 +454068.947}
SPL {X  -159.990, Y  +517.330, Z    +0.000, E1   +22.053, E3 +454078.803}
SPL {X  -159.990, Y  +514.729, Z    +0.000, E1   +22.089, E3 +454092.361}
SPL {X  -159.990, Y  +511.670, Z    +0.000, E1   +22.064, E3 +454108.448}
SPL {X  -159.990, Y  +506.947, Z    +0.000, E1   +23.726, E3 +454118.477}
SPL {X  -159.990, Y  +496.921, Z    +0.000, E1   +28.340, E3 +454127.226}
SPL {X  -159.990, Y  +495.822, Z    +0.000, E1   +27.449, E3 +454137.974}
SPL {X  -159.990, Y  +494.952, Z    +0.000, E1   +26.628, E3 +454147.557}
SPL {X  -159.990, Y  +493.896, Z    +0.000, E1   +25.736, E3 +454158.887}
SPL {X  -159.990, Y  +491.647, Z    +0.000, E1   +25.401, E3 +454171.422}
SPL {X  -159.990, Y  +488.807, Z    +0.000, E1   +25.397, E3 +454184.120}
SPL {X  -159.990, Y  +486.070, Z    +0.000, E1   +25.399, E3 +454196.351}
SPL {X  -159.990, Y  +482.821, Z    +0.000, E1   +25.411, E3 +454210.853}
SPL {X  -159.990, Y  +480.183, Z    +0.000, E1   +25.384, E3 +454222.693}
SPL {X  -159.990, Y  +477.508, Z    +0.000, E1   +25.410, E3 +454234.602}
SPL {X  -159.990, Y  +473.634, Z    +0.000, E1   +25.426, E3 +454251.891}
SPL {X  -159.990, Y  +470.047, Z    +0.000, E1   +25.402, E3 +454267.972}
SPL {X  -159.990, Y  +466.213, Z    +0.000, E1   +25.433, E3 +454285.052}
SPL {X  -159.990, Y  +462.520, Z    +0.000, E1   +25.400, E3 +454301.620}
SPL {X  -159.990, Y  +460.081, Z    +0.000, E1   +25.390, E3 +454312.522}
SPL {X  -159.990, Y  +457.497, Z    +0.000, E1   +25.403, E3 +454324.046}
SPL {X  -159.990, Y  +454.323, Z    +0.000, E1   +25.412, E3 +454338.205}
SPL {X  -159.990, Y  +451.400, Z    +0.000, E1   +25.397, E3 +454351.296}
SPL {X  -159.990, Y  +448.503, Z    +0.000, E1   +25.410, E3 +454364.214}
SPL {X  -159.990, Y  +445.108, Z    +0.000, E1   +25.407, E3 +454379.452}
SPL {X  -159.990, Y  +441.797, Z    +0.000, E1   +25.390, E3 +454394.331}
SPL {X  -159.990, Y  +439.442, Z    +0.000, E1   +25.369, E3 +454404.908}
SPL {X  -159.990, Y  +436.316, Z    +0.000, E1   +25.420, E3 +454418.790}
SPL {X  -159.990, Y  +432.613, Z    +0.000, E1   +25.390, E3 +454435.415}
SPL {X  -159.990, Y  +429.079, Z    +0.000, E1   +25.407, E3 +454451.186}
SPL {X  -159.990, Y  +426.149, Z    +0.000, E1   +25.374, E3 +454464.348}
SPL {X  -159.990, Y  +423.417, Z    +0.000, E1   +25.400, E3 +454476.513}
SPL {X  -159.990, Y  +420.283, Z    +0.000, E1   +25.386, E3 +454490.557}
SPL {X  -159.990, Y  +417.514, Z    +0.000, E1   +25.386, E3 +454502.942}
SPL {X  -159.990, Y  +414.805, Z    +0.000, E1   +25.385, E3 +454515.062}
SPL {X  -159.990, Y  +411.282, Z    +0.000, E1   +25.413, E3 +454530.763}
SPL {X  -159.990, Y  +407.450, Z    +0.000, E1   +25.401, E3 +454547.912}
SPL {X  -159.990, Y  +403.513, Z    +0.000, E1   +25.420, E3 +454565.466}
SPL {X  -159.990, Y  +399.257, Z    +0.000, E1   +25.420, E3 +454584.507}
SPL {X  -159.990, Y  +395.992, Z    +0.000, E1   +25.380, E3 +454599.196}
SPL {X  -159.990, Y  +393.569, Z    +0.000, E1   +25.379, E3 +454610.039}
SPL {X  -159.990, Y  +390.564, Z    +0.000, E1   +25.393, E3 +454623.483}
SPL {X  -159.990, Y  +387.503, Z    +0.000, E1   +25.378, E3 +454637.198}
SPL {X  -159.990, Y  +384.900, Z    +0.000, E1   +25.383, E3 +454648.808}
SPL {X  -159.990, Y  +382.110, Z    +0.000, E1   +25.393, E3 +454661.254}
SPL {X  -159.961, Y  +379.439, Z    +0.000, E1   +25.380, E3 +454673.234}
SPL {X  -159.894, Y  +376.959, Z    +0.000, E1   +25.370, E3 +454684.411}
SPL {X  -159.784, Y  +374.382, Z    +0.000, E1   +25.356, E3 +454696.052}
SPL {X  -159.621, Y  +371.640, Z    +0.000, E1   +25.335, E3 +454708.492}
SPL {X  -159.406, Y  +368.844, Z    +0.000, E1   +25.307, E3 +454721.205}
SPL {X  -159.144, Y  +366.072, Z    +0.000, E1   +25.281, E3 +454733.812}
SPL {X  -158.822, Y  +363.200, Z    +0.000, E1   +25.236, E3 +454746.985}
SPL {X  -158.491, Y  +360.654, Z    +0.000, E1   +25.188, E3 +454758.725}
SPL {X  -158.127, Y  +358.155, Z    +0.000, E1   +25.126, E3 +454770.344}
SPL {X  -158.095, Y  +357.947, Z    +0.000, E1   +21.741, E3 +454801.917}
ENDSPLINE

SPLINE
SPL {X  -158.454, Y  +360.384, Z    +0.000, E1   +19.366, E3 +454814.068}
SPL {X  -159.737, Y  +373.507, Z    +0.000, E1   +10.311, E3 +454836.103}
SPL {X  -159.990, Y  +382.574, Z    +0.000, E1    +4.463, E3 +454842.791}
SPL {X  -159.990, Y  +387.496, Z    +0.000, E1    +1.004, E3 +454845.536}
SPL {X  -159.990, Y  +395.121, Z    +0.000, E1    -4.514, E3 +454849.848}
SPL {X  -159.990, Y  +407.941, Z    +0.000, E1   -14.126, E3 +454861.923}
SPL {X  -159.990, Y  +418.671, Z    +0.000, E1   -19.855, E3 +454881.339}
SPL {X  -159.990, Y  +428.534, Z    +0.000, E1   -23.299, E3 +454904.859}
SPL {X  -159.990, Y  +430.313, Z    +0.000, E1   -23.313, E3 +454913.572}
SPL {X  -159.990, Y  +432.766, Z    +0.000, E1   -23.321, E3 +454925.616}
SPL {X  -159.990, Y  +434.794, Z    +0.000, E1   -23.304, E3 +454935.648}
SPL {X  -159.990, Y  +437.007, Z    +0.000, E1   -23.323, E3 +454946.500}
SPL {X  -159.990, Y  +439.778, Z    +0.000, E1   -23.323, E3 +454960.133}
SPL {X  -159.990, Y  +442.010, Z    +0.000, E1   -23.308, E3 +454971.154}
SPL {X  -159.990, Y  +443.729, Z    +0.000, E1   -23.310, E3 +454979.610}
SPL {X  -159.990, Y  +446.037, Z    +0.000, E1   -23.324, E3 +454990.947}
SPL {X  -159.990, Y  +449.434, Z    +0.000, E1   -23.356, E3 +455007.568}
SPL {X  -159.990, Y  +453.256, Z    +0.000, E1   -23.349, E3 +455026.403}
SPL {X  -159.990, Y  +455.953, Z    +0.000, E1   -23.320, E3 +455039.717}
SPL {X  -159.990, Y  +458.265, Z    +0.000, E1   -23.328, E3 +455051.072}
SPL {X  -159.990, Y  +461.258, Z    +0.000, E1   -23.344, E3 +455065.788}
SPL {X  -159.990, Y  +464.382, Z    +0.000, E1   -23.332, E3 +455081.169}
SPL {X  -159.990, Y  +466.881, Z    +0.000, E1   -23.322, E3 +455093.489}
SPL {X  -159.990, Y  +468.951, Z    +0.000, E1   -23.319, E3 +455103.681}
SPL {X  -159.990, Y  +470.991, Z    +0.000, E1   -23.322, E3 +455113.711}
SPL {X  -159.990, Y  +474.027, Z    +0.000, E1   -23.352, E3 +455128.615}
SPL {X  -159.990, Y  +477.600, Z    +0.000, E1   -23.351, E3 +455146.218}
SPL {X  -159.990, Y  +481.169, Z    +0.000, E1   -23.337, E3 +455163.815}
SPL {X  -159.990, Y  +483.782, Z    +0.000, E1   -23.316, E3 +455176.720}
SPL {X  -159.990, Y  +486.109, Z    +0.000, E1   -23.322, E3 +455188.173}
SPL {X  -159.990, Y  +489.247, Z    +0.000, E1   -23.348, E3 +455203.560}
SPL {X  -159.990, Y  +492.126, Z    +0.000, E1   -23.317, E3 +455217.795}
SPL {X  -159.990, Y  +494.937, Z    +0.000, E1   -23.343, E3 +455231.577}
SPL {X  -159.990, Y  +497.668, Z    +0.000, E1   -23.317, E3 +455245.070}
SPL {X  -159.990, Y  +499.995, Z    +0.000, E1   -23.324, E3 +455256.508}
SPL {X  -159.990, Y  +502.456, Z    +0.000, E1   -23.324, E3 +455268.622}
SPL {X  -159.990, Y  +504.508, Z    +0.000, E1   -23.311, E3 +455278.756}
SPL {X  -159.990, Y  +506.420, Z    +0.000, E1   -23.317, E3 +455288.149}
SPL {X  -159.990, Y  +508.862, Z    +0.000, E1   -23.328, E3 +455300.142}
SPL {X  -159.990, Y  +511.771, Z    +0.000, E1   -23.331, E3 +455314.464}
SPL {X  -159.990, Y  +514.757, Z    +0.000, E1   -23.329, E3 +455329.172}
SPL {X  -159.990, Y  +517.536, Z    +0.000, E1   -23.326, E3 +455342.838}
SPL {X  -159.990, Y  +519.961, Z    +0.000, E1   -23.334, E3 +455354.690}
SPL {X  -159.990, Y  +521.849, Z    +0.000, E1   -23.320, E3 +455364.013}
SPL {X  -159.990, Y  +523.968, Z    +0.000, E1   -23.332, E3 +455374.449}
SPL {X  -159.990, Y  +526.466, Z    +0.000, E1   -23.320, E3 +455386.792}
SPL {X  -159.990, Y  +528.815, Z    +0.000, E1   -23.322, E3 +455398.352}
SPL {X  -159.990, Y  +531.246, Z    +0.000, E1   -23.325, E3 +455410.290}
SPL {X  -159.990, Y  +533.354, Z    +0.000, E1   -23.318, E3 +455420.676}
SPL {X  -159.990, Y  +534.931, Z    +0.000, E1   -23.312, E3 +455428.470}
SPL {X  -159.990, Y  +537.024, Z    +0.000, E1   -23.321, E3 +455438.769}
SPL {X  -159.990, Y  +539.129, Z    +0.000, E1   -23.310, E3 +455449.152}
SPL {X  -159.990, Y  +541.183, Z    +0.000, E1   -23.319, E3 +455459.248}
SPL {X  -159.990, Y  +544.314, Z    +0.000, E1   -23.352, E3 +455474.577}
SPL {X  -159.990, Y  +548.126, Z    +0.000, E1   -23.354, E3 +455493.332}
SPL {X  -159.990, Y  +551.344, Z    +0.000, E1   -23.327, E3 +455509.224}
SPL {X  -159.990, Y  +553.642, Z    +0.000, E1   -23.319, E3 +455520.542}
SPL {X  -159.990, Y  +556.481, Z    +0.000, E1   -23.354, E3 +455534.449}
SPL {X  -159.990, Y  +559.475, Z    +0.000, E1   -23.321, E3 +455549.255}
SPL {X  -159.990, Y  +561.830, Z    +0.000, E1   -23.325, E3 +455560.839}
SPL {X  -159.990, Y  +564.273, Z    +0.000, E1   -23.325, E3 +455572.864}
SPL {X  -159.990, Y  +566.342, Z    +0.000, E1   -23.314, E3 +455583.068}
SPL {X  -159.990, Y  +568.849, Z    +0.000, E1   -23.338, E3 +455595.363}
SPL {X  -159.990, Y  +572.204, Z    +0.000, E1   -23.344, E3 +455611.858}
SPL {X  -159.990, Y  +575.097, Z    +0.000, E1   -23.325, E3 +455626.135}
SPL {X  -159.990, Y  +577.540, Z    +0.000, E1   -23.325, E3 +455638.164}
SPL {X  -159.990, Y  +580.312, Z    +0.000, E1   -23.340, E3 +455651.746}
SPL {X  -159.990, Y  +583.018, Z    +0.000, E1   -23.331, E3 +455665.051}
SPL {X  -159.990, Y  +585.165, Z    +0.000, E1   -23.322, E3 +455675.666}
SPL {X  -159.990, Y  +587.388, Z    +0.000, E1   -23.328, E3 +455686.579}
SPL {X  -159.990, Y  +589.763, Z    +0.000, E1   -23.328, E3 +455698.266}
SPL {X  -159.990, Y  +592.397, Z    +0.000, E1   -23.344, E3 +455711.147}
SPL {X  -159.990, Y  +594.928, Z    +0.000, E1   -23.334, E3 +455723.609}
SPL {X  -159.990, Y  +597.981, Z    +0.000, E1   -23.373, E3 +455738.524}
SPL {X  -159.990, Y  +600.935, Z    +0.000, E1   -23.343, E3 +455753.056}
SPL {X  -159.990, Y  +603.047, Z    +0.000, E1   -23.344, E3 +455763.442}
SPL {X  -159.990, Y  +605.187, Z    +0.000, E1   -23.344, E3 +455773.964}
SPL {X  -159.990, Y  +607.319, Z    +0.000, E1   -23.353, E3 +455784.426}
SPL {X  -159.990, Y  +610.569, Z    +0.000, E1   -23.372, E3 +455800.391}
SPL {X  -159.990, Y  +613.591, Z    +0.000, E1   -23.342, E3 +455815.319}
SPL {X  -159.990, Y  +615.604, Z    +0.000, E1   -23.330, E3 +455825.257}
SPL {X  -159.990, Y  +618.445, Z    +0.000, E1   -23.368, E3 +455839.171}
SPL {X  -159.990, Y  +621.517, Z    +0.000, E1   -23.337, E3 +455854.335}
SPL {X  -159.990, Y  +623.764, Z    +0.000, E1   -23.335, E3 +455865.385}
SPL {X  -159.990, Y  +625.941, Z    +0.000, E1   -23.337, E3 +455876.076}
SPL {X  -159.990, Y  +628.611, Z    +0.000, E1   -23.357, E3 +455889.155}
SPL {X  -159.990, Y  +631.169, Z    +0.000, E1   -23.338, E3 +455901.760}
SPL {X  -159.990, Y  +633.318, Z    +0.000, E1   -23.339, E3 +455912.349}
SPL {X  -159.990, Y  +635.650, Z    +0.000, E1   -23.339, E3 +455923.820}
SPL {X  -159.990, Y  +637.839, Z    +0.000, E1   -23.335, E3 +455934.630}
SPL {X  -159.990, Y  +640.072, Z    +0.000, E1   -23.325, E3 +455945.662}
SPL {X  -159.990, Y  +642.230, Z    +0.000, E1   -23.323, E3 +455956.344}
SPL {X  -159.990, Y  +645.287, Z    +0.000, E1   -23.340, E3 +455971.369}
SPL {X  -159.990, Y  +648.792, Z    +0.000, E1   -23.346, E3 +455988.628}
SPL {X  -159.990, Y  +651.647, Z    +0.000, E1   -23.312, E3 +456002.741}
SPL {X  -159.990, Y  +654.543, Z    +0.000, E1   -23.348, E3 +456016.907}
SPL {X  -159.990, Y  +658.319, Z    +0.000, E1   -23.349, E3 +456035.497}
SPL {X  -159.990, Y  +661.392, Z    +0.000, E1   -23.318, E3 +456050.700}
SPL {X  -159.990, Y  +663.662, Z    +0.000, E1   -23.322, E3 +456061.824}
SPL {X  -159.990, Y  +665.964, Z    +0.000, E1   -23.328, E3 +456073.114}
SPL {X  -159.990, Y  +667.870, Z    +0.000, E1   -23.320, E3 +456082.521}
SPL {X  -159.990, Y  +669.861, Z    +0.000, E1   -23.321, E3 +456092.322}
SPL {X  -159.983, Y  +672.946, Z    +0.000, E1   -23.359, E3 +456107.431}
SPL {X  -159.924, Y  +676.110, Z    +0.000, E1   -23.320, E3 +456123.131}
SPL {X  -159.845, Y  +678.302, Z    +0.000, E1   -23.298, E3 +456134.032}
SPL {X  -159.760, Y  +680.081, Z    +0.000, E1   -23.288, E3 +456142.876}
SPL {X  -159.626, Y  +682.287, Z    +0.000, E1   -23.280, E3 +456153.848}
SPL {X  -159.462, Y  +684.486, Z    +0.000, E1   -23.258, E3 +456164.847}
SPL {X  -159.246, Y  +686.911, Z    +0.000, E1   -23.230, E3 +456177.008}
SPL {X  -159.019, Y  +689.098, Z    +0.000, E1   -23.200, E3 +456188.011}
SPL {X  -158.771, Y  +691.210, Z    +0.000, E1   -23.159, E3 +456198.686}
SPL {X  -158.553, Y  +692.896, Z    +0.000, E1   -23.130, E3 +456207.215}
ENDSPLINE

SPLINE
SPL {X  -159.063, Y  +688.696, Z    +0.000, E1   -17.094, E3 +456245.336}
SPL {X  -159.987, Y  +672.488, Z    +0.000, E1    -5.638, E3 +456269.401}
SPL {X  -159.990, Y  +663.928, Z    +0.000, E1    +0.338, E3 +456275.195}
SPL {X  -159.990, Y  +658.009, Z    +0.000, E1    +4.774, E3 +456278.895}
SPL {X  -159.990, Y  +651.567, Z    +0.000, E1    +9.674, E3 +456284.299}
SPL {X  -159.990, Y  +638.711, Z    +0.000, E1   +17.883, E3 +456299.944}
SPL {X  -159.990, Y  +631.642, Z    +0.000, E1   +20.884, E3 +456315.503}
SPL {X  -159.990, Y  +626.048, Z    +0.000, E1   +22.026, E3 +456335.497}
SPL {X  -159.990, Y  +623.760, Z    +0.000, E1   +22.031, E3 +456347.484}
SPL {X  -159.990, Y  +621.334, Z    +0.000, E1   +22.029, E3 +456360.210}
SPL {X  -159.990, Y  +618.387, Z    +0.000, E1   +22.057, E3 +456375.600}
SPL {X  -159.990, Y  +614.928, Z    +0.000, E1   +22.055, E3 +456393.753}
SPL {X  -159.990, Y  +611.459, Z    +0.000, E1   +22.053, E3 +456411.956}
SPL {X  -159.990, Y  +608.810, Z    +0.000, E1   +22.023, E3 +456425.923}
SPL {X  -159.990, Y  +605.804, Z    +0.000, E1   +22.064, E3 +456441.569}
SPL {X  -159.990, Y  +602.819, Z    +0.000, E1   +22.037, E3 +456457.240}
SPL {X  -159.990, Y  +600.642, Z    +0.000, E1   +22.032, E3 +456468.668}
SPL {X  -159.990, Y  +598.568, Z    +0.000, E1   +22.046, E3 +456479.461}
SPL {X  -159.990, Y  +595.493, Z    +0.000, E1   +22.070, E3 +456495.544}
SPL {X  -159.990, Y  +592.865, Z    +0.000, E1   +22.036, E3 +456509.373}
SPL {X  -159.990, Y  +590.803, Z    +0.000, E1   +22.046, E3 +456520.163}
SPL {X  -159.990, Y  +587.778, Z    +0.000, E1   +22.073, E3 +456535.938}
SPL {X  -159.990, Y  +585.120, Z    +0.000, E1   +22.045, E3 +456549.882}
SPL {X  -159.990, Y  +583.118, Z    +0.000, E1   +22.052, E3 +456560.369}
SPL {X  -159.990, Y  +580.131, Z    +0.000, E1   +22.078, E3 +456575.975}
SPL {X  -159.990, Y  +576.888, Z    +0.000, E1   +22.061, E3 +456593.005}
SPL {X  -159.990, Y  +574.280, Z    +0.000, E1   +22.051, E3 +456606.679}
SPL {X  -159.990, Y  +572.375, Z    +0.000, E1   +22.037, E3 +456616.717}
SPL {X  -159.990, Y  +569.881, Z    +0.000, E1   +22.067, E3 +456629.712}
SPL {X  -159.990, Y  +567.211, Z    +0.000, E1   +22.046, E3 +456643.739}
SPL {X  -159.990, Y  +565.039, Z    +0.000, E1   +22.047, E3 +456655.116}
SPL {X  -159.990, Y  +562.755, Z    +0.000, E1   +22.047, E3 +456667.102}
SPL {X  -159.990, Y  +559.661, Z    +0.000, E1   +22.078, E3 +456683.233}
SPL {X  -159.990, Y  +555.965, Z    +0.000, E1   +22.085, E3 +456702.542}
SPL {X  -159.990, Y  +553.115, Z    +0.000, E1   +22.054, E3 +456717.528}
SPL {X  -159.990, Y  +550.886, Z    +0.000, E1   +22.056, E3 +456729.209}
SPL {X  -159.990, Y  +548.814, Z    +0.000, E1   +22.049, E3 +456740.055}
SPL {X  -159.990, Y  +546.122, Z    +0.000, E1   +22.088, E3 +456754.069}
SPL {X  -159.990, Y  +543.405, Z    +0.000, E1   +22.048, E3 +456768.403}
SPL {X  -159.990, Y  +541.673, Z    +0.000, E1   +22.053, E3 +456777.467}
SPL {X  -159.990, Y  +539.341, Z    +0.000, E1   +22.056, E3 +456789.672}
SPL {X  -159.990, Y  +536.984, Z    +0.000, E1   +22.057, E3 +456802.003}
SPL {X  -159.990, Y  +534.045, Z    +0.000, E1   +22.087, E3 +456817.328}
SPL {X  -159.990, Y  +530.476, Z    +0.000, E1   +22.084, E3 +456836.021}
SPL {X  -159.990, Y  +527.412, Z    +0.000, E1   +22.067, E3 +456852.085}
SPL {X  -159.990, Y  +525.349, Z    +0.000, E1   +22.050, E3 +456862.926}
SPL {X  -159.990, Y  +523.717, Z    +0.000, E1   +22.050, E3 +456871.491}
SPL {X  -159.990, Y  +521.599, Z    +0.000, E1   +22.060, E3 +456882.559}
SPL {X  -159.990, Y  +519.209, Z    +0.000, E1   +22.063, E3 +456895.034}
SPL {X  -159.990, Y  +517.330, Z    +0.000, E1   +22.053, E3 +456904.890}
SPL {X  -159.990, Y  +514.729, Z    +0.000, E1   +22.089, E3 +456918.448}
SPL {X  -159.990, Y  +511.670, Z    +0.000, E1   +22.064, E3 +456934.535}
SPL {X  -159.990, Y  +506.947, Z    +0.000, E1   +23.726, E3 +456944.564}
SPL {X  -159.990, Y  +496.921, Z    +0.000, E1   +28.340, E3 +456953.312}
SPL {X  -159.990, Y  +495.822, Z    +0.000, E1   +27.449, E3 +456964.061}
SPL {X  -159.990, Y  +494.952, Z    +0.000, E1   +26.628, E3 +456973.644}
SPL {X  -159.990, Y  +493.896, Z    +0.000, E1   +25.736, E3 +456984.974}
SPL {X  -159.990, Y  +491.647, Z    +0.000, E1   +25.401, E3 +456997.509}
SPL {X  -159.990, Y  +488.807, Z    +0.000, E1   +25.397, E3 +457010.207}
SPL {X  -159.990, Y  +486.070, Z    +0.000, E1   +25.399, E3 +457022.438}
SPL {X  -159.990, Y  +482.821, Z    +0.000, E1   +25.411, E3 +457036.940}
SPL {X  -159.990, Y  +480.183, Z    +0.000, E1   +25.384, E3 +457048.780}
SPL {X  -159.990, Y  +477.508, Z    +0.000, E1   +25.410, E3 +457060.689}
SPL {X  -159.990, Y  +473.634, Z    +0.000, E1   +25.426, E3 +457077.978}
SPL {X  -159.990, Y  +470.047, Z    +0.000, E1   +25.402, E3 +457094.059}
SPL {X  -159.990, Y  +466.213, Z    +0.000, E1   +25.433, E3 +457111.139}
SPL {X  -159.990, Y  +462.520, Z    +0.000, E1   +25.400, E3 +457127.707}
SPL {X  -159.990, Y  +460.081, Z    +0.000, E1   +25.390, E3 +457138.609}
SPL {X  -159.990, Y  +457.497, Z    +0.000, E1   +25.403, E3 +457150.133}
SPL {X  -159.990, Y  +455.126, Z    +0.000, E1   +25.389, E3 +457160.741}
SPL {X  -159.990, Y  +452.123, Z    +0.000, E1   +25.426, E3 +457174.099}
SPL {X  -159.990, Y  +448.503, Z    +0.000, E1   +25.410, E3 +457190.301}
SPL {X  -159.990, Y  +445.882, Z    +0.000, E1   +25.385, E3 +457202.103}
SPL {X  -159.990, Y  +443.345, Z    +0.000, E1   +25.390, E3 +457213.485}
SPL {X  -159.990, Y  +440.220, Z    +0.000, E1   +25.392, E3 +457227.473}
SPL {X  -159.990, Y  +436.316, Z    +0.000, E1   +25.420, E3 +457244.877}
SPL {X  -159.990, Y  +432.613, Z    +0.000, E1   +25.390, E3 +457261.502}
SPL {X  -159.990, Y  +429.079, Z    +0.000, E1   +25.407, E3 +457277.273}
SPL {X  -159.990, Y  +425.142, Z    +0.000, E1   +25.407, E3 +457294.875}
SPL {X  -159.990, Y  +421.010, Z    +0.000, E1   +25.418, E3 +457313.336}
SPL {X  -159.990, Y  +417.514, Z    +0.000, E1   +25.386, E3 +457329.029}
SPL {X  -159.990, Y  +414.805, Z    +0.000, E1   +25.385, E3 +457341.149}
SPL {X  -159.990, Y  +411.959, Z    +0.000, E1   +25.386, E3 +457353.876}
SPL {X  -159.990, Y  +408.981, Z    +0.000, E1   +25.392, E3 +457367.179}
SPL {X  -159.990, Y  +406.574, Z    +0.000, E1   +25.375, E3 +457377.953}
SPL {X  -159.990, Y  +403.513, Z    +0.000, E1   +25.420, E3 +457391.553}
SPL {X  -159.990, Y  +399.257, Z    +0.000, E1   +25.420, E3 +457410.594}
SPL {X  -159.990, Y  +395.992, Z    +0.000, E1   +25.380, E3 +457425.283}
SPL {X  -159.990, Y  +393.569, Z    +0.000, E1   +25.379, E3 +457436.126}
SPL {X  -159.990, Y  +390.564, Z    +0.000, E1   +25.393, E3 +457449.570}
SPL {X  -159.990, Y  +387.503, Z    +0.000, E1   +25.378, E3 +457463.285}
SPL {X  -159.990, Y  +384.900, Z    +0.000, E1   +25.383, E3 +457474.895}
SPL {X  -159.990, Y  +382.110, Z    +0.000, E1   +25.393, E3 +457487.341}
SPL {X  -159.961, Y  +379.439, Z    +0.000, E1   +25.380, E3 +457499.321}
SPL {X  -159.894, Y  +376.959, Z    +0.000, E1   +25.370, E3 +457510.498}
SPL {X  -159.784, Y  +374.382, Z    +0.000, E1   +25.356, E3 +457522.139}
SPL {X  -159.621, Y  +371.640, Z    +0.000, E1   +25.335, E3 +457534.578}
SPL {X  -159.406, Y  +368.844, Z    +0.000, E1   +25.307, E3 +457547.292}
SPL {X  -159.144, Y  +366.072, Z    +0.000, E1   +25.281, E3 +457559.899}
SPL {X  -158.822, Y  +363.200, Z    +0.000, E1   +25.236, E3 +457573.072}
SPL {X  -158.491, Y  +360.654, Z    +0.000, E1   +25.188, E3 +457584.812}
SPL {X  -158.127, Y  +358.155, Z    +0.000, E1   +25.126, E3 +457596.431}
SPL {X  -158.095, Y  +357.947, Z    +0.000, E1   +21.741, E3 +457628.004}
ENDSPLINE

SPLINE
SPL {X  -158.454, Y  +360.384, Z    +0.000, E1   +19.366, E3 +457640.155}
SPL {X  -159.737, Y  +373.507, Z    +0.000, E1   +10.311, E3 +457662.190}
SPL {X  -159.990, Y  +382.574, Z    +0.000, E1    +4.463, E3 +457668.878}
SPL {X  -159.990, Y  +387.496, Z    +0.000, E1    +1.004, E3 +457671.623}
SPL {X  -159.990, Y  +395.121, Z    +0.000, E1    -4.514, E3 +457675.935}
SPL {X  -159.990, Y  +407.941, Z    +0.000, E1   -14.126, E3 +457688.010}
SPL {X  -159.990, Y  +418.671, Z    +0.000, E1   -19.855, E3 +457707.426}
SPL {X  -159.990, Y  +428.534, Z    +0.000, E1   -23.299, E3 +457730.946}
SPL {X  -159.990, Y  +431.017, Z    +0.000, E1   -23.339, E3 +457743.072}
SPL {X  -159.990, Y  +434.188, Z    +0.000, E1   -23.325, E3 +457758.696}
SPL {X  -159.990, Y  +436.320, Z    +0.000, E1   -23.304, E3 +457769.249}
SPL {X  -159.990, Y  +439.169, Z    +0.000, E1   -23.353, E3 +457783.166}
SPL {X  -159.990, Y  +442.945, Z    +0.000, E1   -23.339, E3 +457801.783}
SPL {X  -159.990, Y  +446.037, Z    +0.000, E1   -23.324, E3 +457817.034}
SPL {X  -159.990, Y  +448.797, Z    +0.000, E1   -23.331, E3 +457830.564}
SPL {X  -159.990, Y  +451.747, Z    +0.000, E1   -23.333, E3 +457845.112}
SPL {X  -159.990, Y  +455.185, Z    +0.000, E1   -23.350, E3 +457861.972}
SPL {X  -159.990, Y  +458.265, Z    +0.000, E1   -23.328, E3 +457877.159}
SPL {X  -159.990, Y  +460.492, Z    +0.000, E1   -23.317, E3 +457888.158}
SPL {X  -159.990, Y  +462.929, Z    +0.000, E1   -23.331, E3 +457900.114}
SPL {X  -159.990, Y  +465.027, Z    +0.000, E1   -23.313, E3 +457910.466}
SPL {X  -159.990, Y  +466.881, Z    +0.000, E1   -23.322, E3 +457919.576}
SPL {X  -159.990, Y  +468.951, Z    +0.000, E1   -23.319, E3 +457929.768}
SPL {X  -159.990, Y  +471.818, Z    +0.000, E1   -23.351, E3 +457943.815}
SPL {X  -159.990, Y  +474.801, Z    +0.000, E1   -23.320, E3 +457958.590}
SPL {X  -159.990, Y  +476.830, Z    +0.000, E1   -23.323, E3 +457968.569}
SPL {X  -159.990, Y  +479.553, Z    +0.000, E1   -23.328, E3 +457981.972}
SPL {X  -159.990, Y  +481.893, Z    +0.000, E1   -23.312, E3 +457993.522}
SPL {X  -159.990, Y  +483.782, Z    +0.000, E1   -23.316, E3 +458002.807}
SPL {X  -159.990, Y  +486.109, Z    +0.000, E1   -23.322, E3 +458014.259}
SPL {X  -159.990, Y  +489.247, Z    +0.000, E1   -23.348, E3 +458029.647}
SPL {X  -159.990, Y  +493.031, Z    +0.000, E1   -23.350, E3 +458048.271}
SPL {X  -159.990, Y  +496.869, Z    +0.000, E1   -23.349, E3 +458067.161}
SPL {X  -159.990, Y  +499.995, Z    +0.000, E1   -23.324, E3 +458082.595}
SPL {X  -159.990, Y  +502.456, Z    +0.000, E1   -23.324, E3 +458094.709}
SPL {X  -159.990, Y  +505.646, Z    +0.000, E1   -23.350, E3 +458110.364}
SPL {X  -159.990, Y  +508.862, Z    +0.000, E1   -23.328, E3 +458126.229}
SPL {X  -159.990, Y  +510.971, Z    +0.000, E1   -23.308, E3 +458136.656}
SPL {X  -159.990, Y  +513.289, Z    +0.000, E1   -23.332, E3 +458148.023}
SPL {X  -159.990, Y  +516.860, Z    +0.000, E1   -23.355, E3 +458165.541}
SPL {X  -159.990, Y  +520.719, Z    +0.000, E1   -23.363, E3 +458184.451}
SPL {X  -159.990, Y  +523.968, Z    +0.000, E1   -23.332, E3 +458200.536}
SPL {X  -159.990, Y  +526.466, Z    +0.000, E1   -23.320, E3 +458212.879}
SPL {X  -159.990, Y  +528.815, Z    +0.000, E1   -23.322, E3 +458224.439}
SPL {X  -159.990, Y  +531.246, Z    +0.000, E1   -23.325, E3 +458236.377}
SPL {X  -159.990, Y  +534.143, Z    +0.000, E1   -23.341, E3 +458250.612}
SPL {X  -159.990, Y  +537.024, Z    +0.000, E1   -23.321, E3 +458264.856}
SPL {X  -159.990, Y  +539.129, Z    +0.000, E1   -23.310, E3 +458275.238}
SPL {X  -159.990, Y  +541.882, Z    +0.000, E1   -23.346, E3 +458288.720}
SPL {X  -159.990, Y  +544.941, Z    +0.000, E1   -23.325, E3 +458303.802}
SPL {X  -159.990, Y  +547.390, Z    +0.000, E1   -23.325, E3 +458315.855}
SPL {X  -159.990, Y  +550.708, Z    +0.000, E1   -23.357, E3 +458332.122}
SPL {X  -159.990, Y  +553.642, Z    +0.000, E1   -23.319, E3 +458346.629}
SPL {X  -159.990, Y  +555.637, Z    +0.000, E1   -23.323, E3 +458356.444}
SPL {X  -159.990, Y  +558.758, Z    +0.000, E1   -23.351, E3 +458371.753}
SPL {X  -159.990, Y  +561.830, Z    +0.000, E1   -23.325, E3 +458386.926}
SPL {X  -159.990, Y  +564.273, Z    +0.000, E1   -23.325, E3 +458398.951}
SPL {X  -159.990, Y  +567.351, Z    +0.000, E1   -23.348, E3 +458414.047}
SPL {X  -159.990, Y  +570.560, Z    +0.000, E1   -23.333, E3 +458429.876}
SPL {X  -159.990, Y  +572.975, Z    +0.000, E1   -23.316, E3 +458441.795}
SPL {X  -159.990, Y  +575.097, Z    +0.000, E1   -23.325, E3 +458452.222}
SPL {X  -159.990, Y  +578.356, Z    +0.000, E1   -23.358, E3 +458468.194}
SPL {X  -159.990, Y  +582.292, Z    +0.000, E1   -23.360, E3 +458487.510}
SPL {X  -159.990, Y  +585.165, Z    +0.000, E1   -23.322, E3 +458501.753}
SPL {X  -159.990, Y  +587.388, Z    +0.000, E1   -23.328, E3 +458512.666}
SPL {X  -159.990, Y  +589.763, Z    +0.000, E1   -23.328, E3 +458524.353}
SPL {X  -159.990, Y  +592.397, Z    +0.000, E1   -23.344, E3 +458537.234}
SPL {X  -159.990, Y  +595.589, Z    +0.000, E1   -23.356, E3 +458552.906}
SPL {X  -159.990, Y  +598.571, Z    +0.000, E1   -23.347, E3 +458567.550}
SPL {X  -159.990, Y  +600.935, Z    +0.000, E1   -23.343, E3 +458579.143}
SPL {X  -159.990, Y  +603.047, Z    +0.000, E1   -23.344, E3 +458589.529}
SPL {X  -159.990, Y  +605.187, Z    +0.000, E1   -23.344, E3 +458600.051}
SPL {X  -159.990, Y  +607.319, Z    +0.000, E1   -23.353, E3 +458610.513}
SPL {X  -159.990, Y  +609.514, Z    +0.000, E1   -23.337, E3 +458621.342}
SPL {X  -159.990, Y  +611.376, Z    +0.000, E1   -23.336, E3 +458630.529}
SPL {X  -159.990, Y  +613.591, Z    +0.000, E1   -23.342, E3 +458641.406}
SPL {X  -159.990, Y  +615.604, Z    +0.000, E1   -23.330, E3 +458651.344}
SPL {X  -159.990, Y  +617.623, Z    +0.000, E1   -23.337, E3 +458661.275}
SPL {X  -159.990, Y  +620.788, Z    +0.000, E1   -23.368, E3 +458676.780}
SPL {X  -159.990, Y  +623.764, Z    +0.000, E1   -23.335, E3 +458691.472}
SPL {X  -159.990, Y  +625.941, Z    +0.000, E1   -23.337, E3 +458702.163}
SPL {X  -159.990, Y  +628.611, Z    +0.000, E1   -23.357, E3 +458715.242}
SPL {X  -159.990, Y  +631.169, Z    +0.000, E1   -23.338, E3 +458727.847}
SPL {X  -159.990, Y  +633.318, Z    +0.000, E1   -23.339, E3 +458738.436}
SPL {X  -159.990, Y  +635.650, Z    +0.000, E1   -23.339, E3 +458749.907}
SPL {X  -159.990, Y  +637.839, Z    +0.000, E1   -23.335, E3 +458760.717}
SPL {X  -159.990, Y  +640.072, Z    +0.000, E1   -23.325, E3 +458771.749}
SPL {X  -159.990, Y  +642.230, Z    +0.000, E1   -23.323, E3 +458782.431}
SPL {X  -159.990, Y  +645.287, Z    +0.000, E1   -23.340, E3 +458797.456}
SPL {X  -159.990, Y  +647.803, Z    +0.000, E1   -23.310, E3 +458809.933}
SPL {X  -159.990, Y  +650.790, Z    +0.000, E1   -23.346, E3 +458824.541}
SPL {X  -159.990, Y  +654.543, Z    +0.000, E1   -23.348, E3 +458842.994}
SPL {X  -159.990, Y  +658.319, Z    +0.000, E1   -23.349, E3 +458861.584}
SPL {X  -159.990, Y  +661.392, Z    +0.000, E1   -23.318, E3 +458876.787}
SPL {X  -159.990, Y  +663.662, Z    +0.000, E1   -23.322, E3 +458887.911}
SPL {X  -159.990, Y  +665.964, Z    +0.000, E1   -23.328, E3 +458899.201}
SPL {X  -159.990, Y  +667.870, Z    +0.000, E1   -23.320, E3 +458908.608}
SPL {X  -159.990, Y  +669.861, Z    +0.000, E1   -23.321, E3 +458918.409}
SPL {X  -159.990, Y  +671.893, Z    +0.000, E1   -23.319, E3 +458928.417}
SPL {X  -159.974, Y  +673.789, Z    +0.000, E1   -23.323, E3 +458937.733}
SPL {X  -159.924, Y  +676.110, Z    +0.000, E1   -23.320, E3 +458949.217}
SPL {X  -159.801, Y  +679.265, Z    +0.000, E1   -23.327, E3 +458964.836}
SPL {X  -159.626, Y  +682.287, Z    +0.000, E1   -23.280, E3 +458979.935}
SPL {X  -159.462, Y  +684.486, Z    +0.000, E1   -23.258, E3 +458990.934}
SPL {X  -159.246, Y  +686.911, Z    +0.000, E1   -23.230, E3 +459003.095}
SPL {X  -159.019, Y  +689.098, Z    +0.000, E1   -23.200, E3 +459014.097}
SPL {X  -158.660, Y  +692.086, Z    +0.000, E1   -23.176, E3 +459029.142}
ENDSPLINE

SPLINE
SPL {X  -159.063, Y  +688.696, Z    +0.000, E1   -17.094, E3 +459071.423}
SPL {X  -159.967, Y  +674.206, Z    +0.000, E1    -6.731, E3 +459094.235}
SPL {X  -159.990, Y  +665.270, Z    +0.000, E1    -0.699, E3 +459100.405}
SPL {X  -159.990, Y  +658.009, Z    +0.000, E1    +4.774, E3 +459104.982}
SPL {X  -159.990, Y  +651.567, Z    +0.000, E1    +9.674, E3 +459110.386}
SPL {X  -159.990, Y  +638.711, Z    +0.000, E1   +17.883, E3 +459126.031}
SPL {X  -159.990, Y  +631.642, Z    +0.000, E1   +20.884, E3 +459141.590}
SPL {X  -159.990, Y  +626.048, Z    +0.000, E1   +22.026, E3 +459161.584}
SPL {X  -159.990, Y  +623.760, Z    +0.000, E1   +22.031, E3 +459173.571}
SPL {X  -159.990, Y  +621.334, Z    +0.000, E1   +22.029, E3 +459186.297}
SPL {X  -159.990, Y  +618.387, Z    +0.000, E1   +22.057, E3 +459201.687}
SPL {X  -159.990, Y  +614.928, Z    +0.000, E1   +22.055, E3 +459219.840}
SPL {X  -159.990, Y  +611.459, Z    +0.000, E1   +22.053, E3 +459238.043}
SPL {X  -159.990, Y  +608.810, Z    +0.000, E1   +22.023, E3 +459252.010}
SPL {X  -159.990, Y  +606.481, Z    +0.000, E1   +22.033, E3 +459264.186}
SPL {X  -159.990, Y  +603.419, Z    +0.000, E1   +22.064, E3 +459280.125}
SPL {X  -159.990, Y  +600.642, Z    +0.000, E1   +22.032, E3 +459294.755}
SPL {X  -159.990, Y  +598.568, Z    +0.000, E1   +22.046, E3 +459305.548}
SPL {X  -159.990, Y  +596.440, Z    +0.000, E1   +22.036, E3 +459316.729}
SPL {X  -159.990, Y  +593.768, Z    +0.000, E1   +22.071, E3 +459330.662}
SPL {X  -159.990, Y  +590.803, Z    +0.000, E1   +22.046, E3 +459346.250}
SPL {X  -159.990, Y  +587.778, Z    +0.000, E1   +22.073, E3 +459362.025}
SPL {X  -159.990, Y  +585.120, Z    +0.000, E1   +22.045, E3 +459375.969}
SPL {X  -159.990, Y  +583.118, Z    +0.000, E1   +22.052, E3 +459386.456}
SPL {X  -159.990, Y  +580.131, Z    +0.000, E1   +22.078, E3 +459402.062}
SPL {X  -159.990, Y  +576.888, Z    +0.000, E1   +22.061, E3 +459419.092}
SPL {X  -159.990, Y  +574.280, Z    +0.000, E1   +22.051, E3 +459432.766}
SPL {X  -159.990, Y  +572.375, Z    +0.000, E1   +22.037, E3 +459442.804}
SPL {X  -159.990, Y  +569.881, Z    +0.000, E1   +22.067, E3 +459455.799}
SPL {X  -159.990, Y  +567.211, Z    +0.000, E1   +22.046, E3 +459469.826}
SPL {X  -159.990, Y  +565.039, Z    +0.000, E1   +22.047, E3 +459481.203}
SPL {X  -159.990, Y  +562.755, Z    +0.000, E1   +22.047, E3 +459493.189}
SPL {X  -159.990, Y  +559.661, Z    +0.000, E1   +22.078, E3 +459509.320}
SPL {X  -159.990, Y  +555.965, Z    +0.000, E1   +22.085, E3 +459528.629}
SPL {X  -159.990, Y  +553.115, Z    +0.000, E1   +22.054, E3 +459543.615}
SPL {X  -159.990, Y  +550.886, Z    +0.000, E1   +22.056, E3 +459555.296}
SPL {X  -159.990, Y  +547.986, Z    +0.000, E1   +22.078, E3 +459570.416}
SPL {X  -159.990, Y  +545.350, Z    +0.000, E1   +22.053, E3 +459584.277}
SPL {X  -159.990, Y  +543.405, Z    +0.000, E1   +22.048, E3 +459594.490}
SPL {X  -159.990, Y  +541.673, Z    +0.000, E1   +22.053, E3 +459603.554}
SPL {X  -159.990, Y  +539.341, Z    +0.000, E1   +22.056, E3 +459615.759}
SPL {X  -159.990, Y  +536.301, Z    +0.000, E1   +22.084, E3 +459631.614}
SPL {X  -159.990, Y  +533.389, Z    +0.000, E1   +22.057, E3 +459646.921}
SPL {X  -159.990, Y  +531.347, Z    +0.000, E1   +22.052, E3 +459657.622}
SPL {X  -159.990, Y  +529.626, Z    +0.000, E1   +22.051, E3 +459666.619}
SPL {X  -159.990, Y  +527.412, Z    +0.000, E1   +22.067, E3 +459678.172}
SPL {X  -159.990, Y  +524.425, Z    +0.000, E1   +22.078, E3 +459693.804}
SPL {X  -159.990, Y  +521.599, Z    +0.000, E1   +22.060, E3 +459708.646}
SPL {X  -159.990, Y  +519.209, Z    +0.000, E1   +22.063, E3 +459721.121}
SPL {X  -159.990, Y  +516.651, Z    +0.000, E1   +22.071, E3 +459734.500}
SPL {X  -159.990, Y  +514.122, Z    +0.000, E1   +22.061, E3 +459747.773}
SPL {X  -159.990, Y  +511.670, Z    +0.000, E1   +22.064, E3 +459760.622}
SPL {X  -159.990, Y  +506.947, Z    +0.000, E1   +23.726, E3 +459770.651}
SPL {X  -159.990, Y  +496.921, Z    +0.000, E1   +28.340, E3 +459779.399}
SPL {X  -159.990, Y  +495.822, Z    +0.000, E1   +27.449, E3 +459790.148}
SPL {X  -159.990, Y  +494.952, Z    +0.000, E1   +26.628, E3 +459799.731}
SPL {X  -159.990, Y  +493.896, Z    +0.000, E1   +25.736, E3 +459811.061}
SPL {X  -159.990, Y  +491.647, Z    +0.000, E1   +25.401, E3 +459823.596}
SPL {X  -159.990, Y  +488.807, Z    +0.000, E1   +25.397, E3 +459836.294}
SPL {X  -159.990, Y  +486.070, Z    +0.000, E1   +25.399, E3 +459848.525}
SPL {X  -159.990, Y  +483.747, Z    +0.000, E1   +25.384, E3 +459858.938}
SPL {X  -159.990, Y  +481.980, Z    +0.000, E1   +25.384, E3 +459866.836}
SPL {X  -159.990, Y  +479.252, Z    +0.000, E1   +25.412, E3 +459878.978}
SPL {X  -159.990, Y  +475.940, Z    +0.000, E1   +25.403, E3 +459893.798}
SPL {X  -159.990, Y  +473.026, Z    +0.000, E1   +25.399, E3 +459906.827}
SPL {X  -159.990, Y  +470.047, Z    +0.000, E1   +25.402, E3 +459920.146}
SPL {X  -159.990, Y  +466.213, Z    +0.000, E1   +25.433, E3 +459937.226}
SPL {X  -159.990, Y  +462.520, Z    +0.000, E1   +25.400, E3 +459953.794}
SPL {X  -159.990, Y  +460.081, Z    +0.000, E1   +25.390, E3 +459964.696}
SPL {X  -159.990, Y  +457.497, Z    +0.000, E1   +25.403, E3 +459976.220}
SPL {X  -159.990, Y  +455.126, Z    +0.000, E1   +25.389, E3 +459986.828}
SPL {X  -159.990, Y  +452.123, Z    +0.000, E1   +25.426, E3 +460000.186}
SPL {X  -159.990, Y  +448.503, Z    +0.000, E1   +25.410, E3 +460016.388}
SPL {X  -159.990, Y  +445.882, Z    +0.000, E1   +25.385, E3 +460028.190}
SPL {X  -159.990, Y  +443.345, Z    +0.000, E1   +25.390, E3 +460039.572}
SPL {X  -159.990, Y  +441.077, Z    +0.000, E1   +25.369, E3 +460049.771}
SPL {X  -159.990, Y  +438.608, Z    +0.000, E1   +25.392, E3 +460060.767}
SPL {X  -159.990, Y  +434.852, Z    +0.000, E1   +25.415, E3 +460077.522}
SPL {X  -159.990, Y  +430.645, Z    +0.000, E1   +25.414, E3 +460096.341}
SPL {X  -159.990, Y  +426.865, Z    +0.000, E1   +25.398, E3 +460113.271}
SPL {X  -159.990, Y  +424.251, Z    +0.000, E1   +25.375, E3 +460125.008}
SPL {X  -159.990, Y  +421.010, Z    +0.000, E1   +25.418, E3 +460139.423}
SPL {X  -159.990, Y  +417.514, Z    +0.000, E1   +25.386, E3 +460155.116}
SPL {X  -159.990, Y  +414.805, Z    +0.000, E1   +25.385, E3 +460167.236}
SPL {X  -159.990, Y  +411.282, Z    +0.000, E1   +25.413, E3 +460182.937}
SPL {X  -159.990, Y  +408.351, Z    +0.000, E1   +25.372, E3 +460196.124}
SPL {X  -159.990, Y  +405.773, Z    +0.000, E1   +25.398, E3 +460207.576}
SPL {X  -159.990, Y  +402.805, Z    +0.000, E1   +25.389, E3 +460220.863}
SPL {X  -159.990, Y  +400.083, Z    +0.000, E1   +25.388, E3 +460233.039}
SPL {X  -159.990, Y  +396.740, Z    +0.000, E1   +25.410, E3 +460247.964}
SPL {X  -159.990, Y  +392.622, Z    +0.000, E1   +25.413, E3 +460266.391}
SPL {X  -159.990, Y  +388.328, Z    +0.000, E1   +25.413, E3 +460285.620}
SPL {X  -159.990, Y  +384.900, Z    +0.000, E1   +25.383, E3 +460300.982}
SPL {X  -159.990, Y  +382.110, Z    +0.000, E1   +25.393, E3 +460313.428}
SPL {X  -159.961, Y  +379.439, Z    +0.000, E1   +25.380, E3 +460325.408}
SPL {X  -159.894, Y  +376.959, Z    +0.000, E1   +25.370, E3 +460336.585}
SPL {X  -159.784, Y  +374.382, Z    +0.000, E1   +25.356, E3 +460348.226}
SPL {X  -159.621, Y  +371.640, Z    +0.000, E1   +25.335, E3 +460360.665}
SPL {X  -159.406, Y  +368.844, Z    +0.000, E1   +25.307, E3 +460373.379}
SPL {X  -159.144, Y  +366.072, Z    +0.000, E1   +25.281, E3 +460385.986}
SPL {X  -158.822, Y  +363.200, Z    +0.000, E1   +25.236, E3 +460399.159}
SPL {X  -158.491, Y  +360.654, Z    +0.000, E1   +25.188, E3 +460410.899}
SPL {X  -158.127, Y  +358.155, Z    +0.000, E1   +25.126, E3 +460422.518}
SPL {X  -158.095, Y  +357.947, Z    +0.000, E1   +21.741, E3 +460454.091}
ENDSPLINE

SPLINE
SPL {X  -158.454, Y  +360.384, Z    +0.000, E1   +19.366, E3 +460466.242}
SPL {X  -159.737, Y  +373.507, Z    +0.000, E1   +10.311, E3 +460488.277}
SPL {X  -159.990, Y  +382.574, Z    +0.000, E1    +4.463, E3 +460494.965}
SPL {X  -159.990, Y  +389.909, Z    +0.000, E1    -0.662, E3 +460498.979}
SPL {X  -159.990, Y  +396.289, Z    +0.000, E1    -5.500, E3 +460502.760}
SPL {X  -159.990, Y  +407.941, Z    +0.000, E1   -14.126, E3 +460514.097}
SPL {X  -159.990, Y  +418.671, Z    +0.000, E1   -19.855, E3 +460533.513}
SPL {X  -159.990, Y  +429.878, Z    +0.000, E1   -23.330, E3 +460563.568}
SPL {X  -159.990, Y  +432.103, Z    +0.000, E1   -23.301, E3 +460574.586}
SPL {X  -159.990, Y  +434.188, Z    +0.000, E1   -23.325, E3 +460584.783}
SPL {X  -159.990, Y  +437.007, Z    +0.000, E1   -23.323, E3 +460598.674}
SPL {X  -159.990, Y  +439.778, Z    +0.000, E1   -23.323, E3 +460612.306}
SPL {X  -159.990, Y  +442.945, Z    +0.000, E1   -23.339, E3 +460627.870}
SPL {X  -159.990, Y  +446.037, Z    +0.000, E1   -23.324, E3 +460643.121}
SPL {X  -159.990, Y  +448.797, Z    +0.000, E1   -23.331, E3 +460656.651}
SPL {X  -159.990, Y  +451.747, Z    +0.000, E1   -23.333, E3 +460671.199}
SPL {X  -159.990, Y  +454.210, Z    +0.000, E1   -23.316, E3 +460683.330}
SPL {X  -159.990, Y  +455.953, Z    +0.000, E1   -23.320, E3 +460691.891}
SPL {X  -159.990, Y  +458.265, Z    +0.000, E1   -23.328, E3 +460703.246}
SPL {X  -159.990, Y  +461.258, Z    +0.000, E1   -23.344, E3 +460717.962}
SPL {X  -159.990, Y  +464.382, Z    +0.000, E1   -23.332, E3 +460733.343}
SPL {X  -159.990, Y  +466.881, Z    +0.000, E1   -23.322, E3 +460745.663}
SPL {X  -159.990, Y  +468.951, Z    +0.000, E1   -23.319, E3 +460755.855}
SPL {X  -159.990, Y  +470.991, Z    +0.000, E1   -23.322, E3 +460765.885}
SPL {X  -159.990, Y  +474.027, Z    +0.000, E1   -23.352, E3 +460780.789}
SPL {X  -159.990, Y  +477.600, Z    +0.000, E1   -23.351, E3 +460798.392}
SPL {X  -159.990, Y  +481.169, Z    +0.000, E1   -23.337, E3 +460815.989}
SPL {X  -159.990, Y  +483.782, Z    +0.000, E1   -23.316, E3 +460828.894}
SPL {X  -159.990, Y  +486.109, Z    +0.000, E1   -23.322, E3 +460840.346}
SPL {X  -159.990, Y  +489.247, Z    +0.000, E1   -23.348, E3 +460855.734}
SPL {X  -159.990, Y  +493.031, Z    +0.000, E1   -23.350, E3 +460874.358}
SPL {X  -159.990, Y  +496.869, Z    +0.000, E1   -23.349, E3 +460893.248}
SPL {X  -159.990, Y  +499.995, Z    +0.000, E1   -23.324, E3 +460908.682}
SPL {X  -159.990, Y  +502.456, Z    +0.000, E1   -23.324, E3 +460920.796}
SPL {X  -159.990, Y  +505.646, Z    +0.000, E1   -23.350, E3 +460936.451}
SPL {X  -159.990, Y  +508.862, Z    +0.000, E1   -23.328, E3 +460952.316}
SPL {X  -159.990, Y  +510.971, Z    +0.000, E1   -23.308, E3 +460962.743}
SPL {X  -159.990, Y  +513.289, Z    +0.000, E1   -23.332, E3 +460974.110}
SPL {X  -159.990, Y  +516.860, Z    +0.000, E1   -23.355, E3 +460991.627}
SPL {X  -159.990, Y  +520.719, Z    +0.000, E1   -23.363, E3 +461010.538}
SPL {X  -159.990, Y  +523.968, Z    +0.000, E1   -23.332, E3 +461026.623}
SPL {X  -159.990, Y  +526.466, Z    +0.000, E1   -23.320, E3 +461038.966}
SPL {X  -159.990, Y  +528.815, Z    +0.000, E1   -23.322, E3 +461050.525}
SPL {X  -159.990, Y  +531.246, Z    +0.000, E1   -23.325, E3 +461062.464}
SPL {X  -159.990, Y  +534.143, Z    +0.000, E1   -23.341, E3 +461076.699}
SPL {X  -159.990, Y  +537.024, Z    +0.000, E1   -23.321, E3 +461090.943}
SPL {X  -159.990, Y  +539.129, Z    +0.000, E1   -23.310, E3 +461101.325}
SPL {X  -159.990, Y  +541.882, Z    +0.000, E1   -23.346, E3 +461114.807}
SPL {X  -159.990, Y  +544.941, Z    +0.000, E1   -23.325, E3 +461129.889}
SPL {X  -159.990, Y  +547.390, Z    +0.000, E1   -23.325, E3 +461141.942}
SPL {X  -159.990, Y  +550.708, Z    +0.000, E1   -23.357, E3 +461158.209}
SPL {X  -159.990, Y  +553.642, Z    +0.000, E1   -23.319, E3 +461172.716}
SPL {X  -159.990, Y  +555.637, Z    +0.000, E1   -23.323, E3 +461182.531}
SPL {X  -159.990, Y  +558.758, Z    +0.000, E1   -23.351, E3 +461197.840}
SPL {X  -159.990, Y  +561.830, Z    +0.000, E1   -23.325, E3 +461213.013}
SPL {X  -159.990, Y  +564.273, Z    +0.000, E1   -23.325, E3 +461225.038}
SPL {X  -159.990, Y  +567.351, Z    +0.000, E1   -23.348, E3 +461240.134}
SPL {X  -159.990, Y  +570.560, Z    +0.000, E1   -23.333, E3 +461255.963}
SPL {X  -159.990, Y  +572.975, Z    +0.000, E1   -23.316, E3 +461267.882}
SPL {X  -159.990, Y  +575.097, Z    +0.000, E1   -23.325, E3 +461278.309}
SPL {X  -159.990, Y  +578.356, Z    +0.000, E1   -23.358, E3 +461294.281}
SPL {X  -159.990, Y  +582.292, Z    +0.000, E1   -23.360, E3 +461313.597}
SPL {X  -159.990, Y  +585.165, Z    +0.000, E1   -23.322, E3 +461327.840}
SPL {X  -159.990, Y  +587.388, Z    +0.000, E1   -23.328, E3 +461338.753}
SPL {X  -159.990, Y  +590.594, Z    +0.000, E1   -23.363, E3 +461354.445}
SPL {X  -159.990, Y  +594.301, Z    +0.000, E1   -23.358, E3 +461372.650}
SPL {X  -159.990, Y  +597.981, Z    +0.000, E1   -23.373, E3 +461390.697}
SPL {X  -159.990, Y  +600.935, Z    +0.000, E1   -23.343, E3 +461405.230}
SPL {X  -159.990, Y  +603.047, Z    +0.000, E1   -23.344, E3 +461415.616}
SPL {X  -159.990, Y  +605.187, Z    +0.000, E1   -23.344, E3 +461426.138}
SPL {X  -159.990, Y  +607.319, Z    +0.000, E1   -23.353, E3 +461436.600}
SPL {X  -159.990, Y  +610.569, Z    +0.000, E1   -23.372, E3 +461452.565}
SPL {X  -159.990, Y  +613.591, Z    +0.000, E1   -23.342, E3 +461467.493}
SPL {X  -159.990, Y  +615.604, Z    +0.000, E1   -23.330, E3 +461477.431}
SPL {X  -159.990, Y  +617.623, Z    +0.000, E1   -23.337, E3 +461487.362}
SPL {X  -159.990, Y  +620.788, Z    +0.000, E1   -23.368, E3 +461502.867}
SPL {X  -159.990, Y  +623.764, Z    +0.000, E1   -23.335, E3 +461517.559}
SPL {X  -159.990, Y  +625.941, Z    +0.000, E1   -23.337, E3 +461528.250}
SPL {X  -159.990, Y  +628.611, Z    +0.000, E1   -23.357, E3 +461541.329}
SPL {X  -159.990, Y  +631.169, Z    +0.000, E1   -23.338, E3 +461553.934}
SPL {X  -159.990, Y  +633.318, Z    +0.000, E1   -23.339, E3 +461564.523}
SPL {X  -159.990, Y  +635.650, Z    +0.000, E1   -23.339, E3 +461575.994}
SPL {X  -159.990, Y  +637.839, Z    +0.000, E1   -23.335, E3 +461586.804}
SPL {X  -159.990, Y  +640.072, Z    +0.000, E1   -23.325, E3 +461597.836}
SPL {X  -159.990, Y  +642.230, Z    +0.000, E1   -23.323, E3 +461608.518}
SPL {X  -159.990, Y  +645.287, Z    +0.000, E1   -23.340, E3 +461623.543}
SPL {X  -159.990, Y  +648.792, Z    +0.000, E1   -23.346, E3 +461640.802}
SPL {X  -159.990, Y  +652.623, Z    +0.000, E1   -23.348, E3 +461659.637}
SPL {X  -159.990, Y  +656.380, Z    +0.000, E1   -23.347, E3 +461678.132}
SPL {X  -159.990, Y  +659.180, Z    +0.000, E1   -23.314, E3 +461691.980}
SPL {X  -159.990, Y  +661.392, Z    +0.000, E1   -23.318, E3 +461702.874}
SPL {X  -159.990, Y  +663.662, Z    +0.000, E1   -23.322, E3 +461713.998}
SPL {X  -159.990, Y  +665.964, Z    +0.000, E1   -23.328, E3 +461725.288}
SPL {X  -159.990, Y  +668.989, Z    +0.000, E1   -23.359, E3 +461740.124}
SPL {X  -159.983, Y  +672.946, Z    +0.000, E1   -23.359, E3 +461759.605}
SPL {X  -159.924, Y  +676.110, Z    +0.000, E1   -23.320, E3 +461775.304}
SPL {X  -159.845, Y  +678.302, Z    +0.000, E1   -23.298, E3 +461786.206}
SPL {X  -159.760, Y  +680.081, Z    +0.000, E1   -23.288, E3 +461795.050}
SPL {X  -159.626, Y  +682.287, Z    +0.000, E1   -23.280, E3 +461806.022}
SPL {X  -159.462, Y  +684.486, Z    +0.000, E1   -23.258, E3 +461817.021}
SPL {X  -159.246, Y  +686.911, Z    +0.000, E1   -23.230, E3 +461829.182}
SPL {X  -159.019, Y  +689.098, Z    +0.000, E1   -23.200, E3 +461840.184}
SPL {X  -158.660, Y  +692.086, Z    +0.000, E1   -23.176, E3 +461855.229}
ENDSPLINE

SPLINE
SPL {X  -159.063, Y  +688.696, Z    +0.000, E1   -17.094, E3 +461897.510}
SPL {X  -159.967, Y  +674.206, Z    +0.000, E1    -6.731, E3 +461920.322}
SPL {X  -159.990, Y  +665.270, Z    +0.000, E1    -0.699, E3 +461926.492}
SPL {X  -159.990, Y  +658.009, Z    +0.000, E1    +4.774, E3 +461931.069}
SPL {X  -159.990, Y  +651.567, Z    +0.000, E1    +9.674, E3 +461936.473}
SPL {X  -159.990, Y  +638.711, Z    +0.000, E1   +17.883, E3 +461952.118}
SPL {X  -159.990, Y  +631.642, Z    +0.000, E1   +20.884, E3 +461967.677}
SPL {X  -159.990, Y  +626.048, Z    +0.000, E1   +22.026, E3 +461987.670}
SPL {X  -159.990, Y  +623.760, Z    +0.000, E1   +22.031, E3 +461999.658}
SPL {X  -159.990, Y  +621.334, Z    +0.000, E1   +22.029, E3 +462012.384}
SPL {X  -159.990, Y  +619.505, Z    +0.000, E1   +22.018, E3 +462022.000}
SPL {X  -159.990, Y  +617.621, Z    +0.000, E1   +22.025, E3 +462031.865}
SPL {X  -159.990, Y  +615.830, Z    +0.000, E1   +22.023, E3 +462041.265}
SPL {X  -159.990, Y  +614.007, Z    +0.000, E1   +22.018, E3 +462050.843}
SPL {X  -159.990, Y  +611.459, Z    +0.000, E1   +22.053, E3 +462064.130}
SPL {X  -159.990, Y  +608.810, Z    +0.000, E1   +22.023, E3 +462078.097}
SPL {X  -159.990, Y  +606.481, Z    +0.000, E1   +22.033, E3 +462090.273}
SPL {X  -159.990, Y  +603.419, Z    +0.000, E1   +22.064, E3 +462106.212}
SPL {X  -159.990, Y  +600.642, Z    +0.000, E1   +22.032, E3 +462120.842}
SPL {X  -159.990, Y  +598.568, Z    +0.000, E1   +22.046, E3 +462131.635}
SPL {X  -159.990, Y  +595.493, Z    +0.000, E1   +22.070, E3 +462147.718}
SPL {X  -159.990, Y  +592.865, Z    +0.000, E1   +22.036, E3 +462161.546}
SPL {X  -159.990, Y  +590.803, Z    +0.000, E1   +22.046, E3 +462172.337}
SPL {X  -159.990, Y  +587.778, Z    +0.000, E1   +22.073, E3 +462188.112}
SPL {X  -159.990, Y  +585.120, Z    +0.000, E1   +22.045, E3 +462202.056}
SPL {X  -159.990, Y  +583.118, Z    +0.000, E1   +22.052, E3 +462212.543}
SPL {X  -159.990, Y  +580.131, Z    +0.000, E1   +22.078, E3 +462228.149}
SPL {X  -159.990, Y  +576.888, Z    +0.000, E1   +22.061, E3 +462245.179}
SPL {X  -159.990, Y  +574.280, Z    +0.000, E1   +22.051, E3 +462258.853}
SPL {X  -159.990, Y  +572.375, Z    +0.000, E1   +22.037, E3 +462268.891}
SPL {X  -159.990, Y  +569.881, Z    +0.000, E1   +22.067, E3 +462281.886}
SPL {X  -159.990, Y  +567.211, Z    +0.000, E1   +22.046, E3 +462295.913}
SPL {X  -159.990, Y  +565.039, Z    +0.000, E1   +22.047, E3 +462307.290}
SPL {X  -159.990, Y  +562.755, Z    +0.000, E1   +22.047, E3 +462319.276}
SPL {X  -159.990, Y  +560.652, Z    +0.000, E1   +22.038, E3 +462330.321}
SPL {X  -159.990, Y  +558.852, Z    +0.000, E1   +22.046, E3 +462339.692}
SPL {X  -159.990, Y  +556.672, Z    +0.000, E1   +22.055, E3 +462351.082}
SPL {X  -159.990, Y  +553.726, Z    +0.000, E1   +22.080, E3 +462366.444}
SPL {X  -159.990, Y  +550.886, Z    +0.000, E1   +22.056, E3 +462381.383}
SPL {X  -159.990, Y  +548.814, Z    +0.000, E1   +22.049, E3 +462392.229}
SPL {X  -159.990, Y  +546.122, Z    +0.000, E1   +22.088, E3 +462406.243}
SPL {X  -159.990, Y  +542.390, Z    +0.000, E1   +22.086, E3 +462425.825}
SPL {X  -159.990, Y  +539.341, Z    +0.000, E1   +22.056, E3 +462441.846}
SPL {X  -159.990, Y  +536.984, Z    +0.000, E1   +22.057, E3 +462454.177}
SPL {X  -159.990, Y  +534.045, Z    +0.000, E1   +22.087, E3 +462469.502}
SPL {X  -159.990, Y  +530.476, Z    +0.000, E1   +22.084, E3 +462488.195}
SPL {X  -159.990, Y  +527.412, Z    +0.000, E1   +22.067, E3 +462504.259}
SPL {X  -159.990, Y  +524.425, Z    +0.000, E1   +22.078, E3 +462519.891}
SPL {X  -159.990, Y  +521.599, Z    +0.000, E1   +22.060, E3 +462534.733}
SPL {X  -159.990, Y  +519.209, Z    +0.000, E1   +22.063, E3 +462547.208}
SPL {X  -159.990, Y  +516.651, Z    +0.000, E1   +22.071, E3 +462560.587}
SPL {X  -159.990, Y  +514.122, Z    +0.000, E1   +22.061, E3 +462573.860}
SPL {X  -159.990, Y  +511.670, Z    +0.000, E1   +22.064, E3 +462586.709}
SPL {X  -159.990, Y  +506.947, Z    +0.000, E1   +23.726, E3 +462596.738}
SPL {X  -159.990, Y  +496.921, Z    +0.000, E1   +28.340, E3 +462605.486}
SPL {X  -159.990, Y  +495.822, Z    +0.000, E1   +27.449, E3 +462616.235}
SPL {X  -159.990, Y  +494.952, Z    +0.000, E1   +26.628, E3 +462625.818}
SPL {X  -159.990, Y  +493.896, Z    +0.000, E1   +25.736, E3 +462637.147}
SPL {X  -159.990, Y  +491.647, Z    +0.000, E1   +25.401, E3 +462649.683}
SPL {X  -159.990, Y  +488.807, Z    +0.000, E1   +25.397, E3 +462662.381}
SPL {X  -159.990, Y  +486.070, Z    +0.000, E1   +25.399, E3 +462674.612}
SPL {X  -159.990, Y  +483.747, Z    +0.000, E1   +25.384, E3 +462685.025}
SPL {X  -159.990, Y  +481.980, Z    +0.000, E1   +25.384, E3 +462692.923}
SPL {X  -159.990, Y  +479.252, Z    +0.000, E1   +25.412, E3 +462705.064}
SPL {X  -159.990, Y  +475.940, Z    +0.000, E1   +25.403, E3 +462719.885}
SPL {X  -159.990, Y  +473.026, Z    +0.000, E1   +25.399, E3 +462732.914}
SPL {X  -159.990, Y  +470.047, Z    +0.000, E1   +25.402, E3 +462746.233}
SPL {X  -159.990, Y  +466.213, Z    +0.000, E1   +25.433, E3 +462763.313}
SPL {X  -159.990, Y  +462.520, Z    +0.000, E1   +25.400, E3 +462779.881}
SPL {X  -159.990, Y  +460.081, Z    +0.000, E1   +25.390, E3 +462790.783}
SPL {X  -159.990, Y  +457.497, Z    +0.000, E1   +25.403, E3 +462802.307}
SPL {X  -159.990, Y  +455.126, Z    +0.000, E1   +25.389, E3 +462812.915}
SPL {X  -159.990, Y  +452.123, Z    +0.000, E1   +25.426, E3 +462826.273}
SPL {X  -159.990, Y  +448.503, Z    +0.000, E1   +25.410, E3 +462842.475}
SPL {X  -159.990, Y  +445.882, Z    +0.000, E1   +25.385, E3 +462854.277}
SPL {X  -159.990, Y  +443.345, Z    +0.000, E1   +25.390, E3 +462865.659}
SPL {X  -159.990, Y  +441.077, Z    +0.000, E1   +25.369, E3 +462875.858}
SPL {X  -159.990, Y  +438.608, Z    +0.000, E1   +25.392, E3 +462886.854}
SPL {X  -159.990, Y  +435.579, Z    +0.000, E1   +25.386, E3 +462900.408}
SPL {X  -159.990, Y  +432.613, Z    +0.000, E1   +25.390, E3 +462913.676}
SPL {X  -159.990, Y  +429.079, Z    +0.000, E1   +25.407, E3 +462929.446}
SPL {X  -159.990, Y  +426.149, Z    +0.000, E1   +25.374, E3 +462942.609}
SPL {X  -159.990, Y  +423.417, Z    +0.000, E1   +25.400, E3 +462954.774}
SPL {X  -159.990, Y  +420.283, Z    +0.000, E1   +25.386, E3 +462968.818}
SPL {X  -159.990, Y  +417.514, Z    +0.000, E1   +25.386, E3 +462981.203}
SPL {X  -159.990, Y  +414.805, Z    +0.000, E1   +25.385, E3 +462993.323}
SPL {X  -159.990, Y  +411.282, Z    +0.000, E1   +25.413, E3 +463009.024}
SPL {X  -159.990, Y  +408.351, Z    +0.000, E1   +25.372, E3 +463022.211}
SPL {X  -159.990, Y  +405.773, Z    +0.000, E1   +25.398, E3 +463033.663}
SPL {X  -159.990, Y  +402.805, Z    +0.000, E1   +25.389, E3 +463046.950}
SPL {X  -159.990, Y  +400.083, Z    +0.000, E1   +25.388, E3 +463059.126}
SPL {X  -159.990, Y  +396.740, Z    +0.000, E1   +25.410, E3 +463074.051}
SPL {X  -159.990, Y  +392.622, Z    +0.000, E1   +25.413, E3 +463092.478}
SPL {X  -159.990, Y  +388.328, Z    +0.000, E1   +25.413, E3 +463111.707}
SPL {X  -159.990, Y  +384.900, Z    +0.000, E1   +25.383, E3 +463127.069}
SPL {X  -159.990, Y  +382.110, Z    +0.000, E1   +25.393, E3 +463139.515}
SPL {X  -159.961, Y  +379.439, Z    +0.000, E1   +25.380, E3 +463151.495}
SPL {X  -159.894, Y  +376.959, Z    +0.000, E1   +25.370, E3 +463162.672}
SPL {X  -159.784, Y  +374.382, Z    +0.000, E1   +25.356, E3 +463174.312}
SPL {X  -159.621, Y  +371.640, Z    +0.000, E1   +25.335, E3 +463186.752}
SPL {X  -159.406, Y  +368.844, Z    +0.000, E1   +25.307, E3 +463199.466}
SPL {X  -159.144, Y  +366.072, Z    +0.000, E1   +25.281, E3 +463212.073}
SPL {X  -158.822, Y  +363.200, Z    +0.000, E1   +25.236, E3 +463225.246}
SPL {X  -158.491, Y  +360.654, Z    +0.000, E1   +25.188, E3 +463236.986}
SPL {X  -158.127, Y  +358.155, Z    +0.000, E1   +25.126, E3 +463248.605}
SPL {X  -158.095, Y  +357.947, Z    +0.000, E1   +21.741, E3 +463280.178}
ENDSPLINE

SPLINE
SPL {X  -158.454, Y  +360.384, Z    +0.000, E1   +19.366, E3 +463292.329}
SPL {X  -159.737, Y  +373.507, Z    +0.000, E1   +10.311, E3 +463314.364}
SPL {X  -159.990, Y  +382.574, Z    +0.000, E1    +4.463, E3 +463321.052}
SPL {X  -159.990, Y  +387.496, Z    +0.000, E1    +1.004, E3 +463323.797}
SPL {X  -159.990, Y  +395.121, Z    +0.000, E1    -4.514, E3 +463328.109}
SPL {X  -159.990, Y  +407.941, Z    +0.000, E1   -14.126, E3 +463340.183}
SPL {X  -159.990, Y  +418.671, Z    +0.000, E1   -19.855, E3 +463359.600}
SPL {X  -159.990, Y  +429.878, Z    +0.000, E1   -23.330, E3 +463389.655}
SPL {X  -159.990, Y  +432.766, Z    +0.000, E1   -23.321, E3 +463403.877}
SPL {X  -159.990, Y  +434.794, Z    +0.000, E1   -23.304, E3 +463413.909}
SPL {X  -159.990, Y  +437.007, Z    +0.000, E1   -23.323, E3 +463424.761}
SPL {X  -159.990, Y  +439.778, Z    +0.000, E1   -23.323, E3 +463438.393}
SPL {X  -159.990, Y  +442.010, Z    +0.000, E1   -23.308, E3 +463449.414}
SPL {X  -159.990, Y  +443.729, Z    +0.000, E1   -23.310, E3 +463457.871}
SPL {X  -159.990, Y  +446.037, Z    +0.000, E1   -23.324, E3 +463469.208}
SPL {X  -159.990, Y  +448.797, Z    +0.000, E1   -23.331, E3 +463482.738}
SPL {X  -159.990, Y  +451.747, Z    +0.000, E1   -23.333, E3 +463497.286}
SPL {X  -159.990, Y  +455.185, Z    +0.000, E1   -23.350, E3 +463514.146}
SPL {X  -159.990, Y  +458.265, Z    +0.000, E1   -23.328, E3 +463529.333}
SPL {X  -159.990, Y  +460.492, Z    +0.000, E1   -23.317, E3 +463540.332}
SPL {X  -159.990, Y  +462.929, Z    +0.000, E1   -23.331, E3 +463552.288}
SPL {X  -159.990, Y  +465.027, Z    +0.000, E1   -23.313, E3 +463562.640}
SPL {X  -159.990, Y  +466.881, Z    +0.000, E1   -23.322, E3 +463571.750}
SPL {X  -159.990, Y  +468.951, Z    +0.000, E1   -23.319, E3 +463581.942}
SPL {X  -159.990, Y  +471.818, Z    +0.000, E1   -23.351, E3 +463595.989}
SPL {X  -159.990, Y  +474.801, Z    +0.000, E1   -23.320, E3 +463610.764}
SPL {X  -159.990, Y  +476.830, Z    +0.000, E1   -23.323, E3 +463620.743}
SPL {X  -159.990, Y  +479.553, Z    +0.000, E1   -23.328, E3 +463634.146}
SPL {X  -159.990, Y  +482.950, Z    +0.000, E1   -23.350, E3 +463650.818}
SPL {X  -159.990, Y  +486.109, Z    +0.000, E1   -23.322, E3 +463666.433}
SPL {X  -159.990, Y  +488.481, Z    +0.000, E1   -23.319, E3 +463678.113}
SPL {X  -159.990, Y  +491.454, Z    +0.000, E1   -23.343, E3 +463692.693}
SPL {X  -159.990, Y  +494.937, Z    +0.000, E1   -23.343, E3 +463709.838}
SPL {X  -159.990, Y  +497.668, Z    +0.000, E1   -23.317, E3 +463723.331}
SPL {X  -159.990, Y  +499.995, Z    +0.000, E1   -23.324, E3 +463734.769}
SPL {X  -159.990, Y  +502.456, Z    +0.000, E1   -23.324, E3 +463746.883}
SPL {X  -159.990, Y  +505.646, Z    +0.000, E1   -23.350, E3 +463762.538}
SPL {X  -159.990, Y  +508.862, Z    +0.000, E1   -23.328, E3 +463778.403}
SPL {X  -159.990, Y  +510.971, Z    +0.000, E1   -23.308, E3 +463788.830}
SPL {X  -159.990, Y  +513.289, Z    +0.000, E1   -23.332, E3 +463800.197}
SPL {X  -159.990, Y  +516.860, Z    +0.000, E1   -23.355, E3 +463817.714}
SPL {X  -159.990, Y  +520.719, Z    +0.000, E1   -23.363, E3 +463836.625}
SPL {X  -159.990, Y  +523.968, Z    +0.000, E1   -23.332, E3 +463852.710}
SPL {X  -159.990, Y  +526.466, Z    +0.000, E1   -23.320, E3 +463865.053}
SPL {X  -159.990, Y  +528.815, Z    +0.000, E1   -23.322, E3 +463876.612}
SPL {X  -159.990, Y  +531.246, Z    +0.000, E1   -23.325, E3 +463888.551}
SPL {X  -159.990, Y  +534.143, Z    +0.000, E1   -23.341, E3 +463902.786}
SPL {X  -159.990, Y  +537.024, Z    +0.000, E1   -23.321, E3 +463917.029}
SPL {X  -159.990, Y  +539.129, Z    +0.000, E1   -23.310, E3 +463927.412}
SPL {X  -159.990, Y  +541.882, Z    +0.000, E1   -23.346, E3 +463940.893}
SPL {X  -159.990, Y  +544.941, Z    +0.000, E1   -23.325, E3 +463955.976}
SPL {X  -159.990, Y  +547.390, Z    +0.000, E1   -23.325, E3 +463968.029}
SPL {X  -159.990, Y  +550.708, Z    +0.000, E1   -23.357, E3 +463984.296}
SPL {X  -159.990, Y  +553.642, Z    +0.000, E1   -23.319, E3 +463998.803}
SPL {X  -159.990, Y  +555.637, Z    +0.000, E1   -23.323, E3 +464008.618}
SPL {X  -159.990, Y  +558.758, Z    +0.000, E1   -23.351, E3 +464023.927}
SPL {X  -159.990, Y  +561.830, Z    +0.000, E1   -23.325, E3 +464039.100}
SPL {X  -159.990, Y  +564.273, Z    +0.000, E1   -23.325, E3 +464051.125}
SPL {X  -159.990, Y  +567.351, Z    +0.000, E1   -23.348, E3 +464066.220}
SPL {X  -159.990, Y  +570.560, Z    +0.000, E1   -23.333, E3 +464082.050}
SPL {X  -159.990, Y  +572.975, Z    +0.000, E1   -23.316, E3 +464093.969}
SPL {X  -159.990, Y  +575.097, Z    +0.000, E1   -23.325, E3 +464104.396}
SPL {X  -159.990, Y  +578.356, Z    +0.000, E1   -23.358, E3 +464120.368}
SPL {X  -159.990, Y  +582.292, Z    +0.000, E1   -23.360, E3 +464139.684}
SPL {X  -159.990, Y  +585.165, Z    +0.000, E1   -23.322, E3 +464153.927}
SPL {X  -159.990, Y  +587.388, Z    +0.000, E1   -23.328, E3 +464164.840}
SPL {X  -159.990, Y  +589.763, Z    +0.000, E1   -23.328, E3 +464176.527}
SPL {X  -159.990, Y  +592.397, Z    +0.000, E1   -23.344, E3 +464189.408}
SPL {X  -159.990, Y  +595.589, Z    +0.000, E1   -23.356, E3 +464205.080}
SPL {X  -159.990, Y  +598.571, Z    +0.000, E1   -23.347, E3 +464219.724}
SPL {X  -159.990, Y  +600.935, Z    +0.000, E1   -23.343, E3 +464231.317}
SPL {X  -159.990, Y  +603.047, Z    +0.000, E1   -23.344, E3 +464241.703}
SPL {X  -159.990, Y  +605.187, Z    +0.000, E1   -23.344, E3 +464252.224}
SPL {X  -159.990, Y  +607.319, Z    +0.000, E1   -23.353, E3 +464262.687}
SPL {X  -159.990, Y  +609.514, Z    +0.000, E1   -23.337, E3 +464273.516}
SPL {X  -159.990, Y  +611.376, Z    +0.000, E1   -23.336, E3 +464282.703}
SPL {X  -159.990, Y  +613.591, Z    +0.000, E1   -23.342, E3 +464293.580}
SPL {X  -159.990, Y  +615.604, Z    +0.000, E1   -23.330, E3 +464303.518}
SPL {X  -159.990, Y  +617.623, Z    +0.000, E1   -23.337, E3 +464313.448}
SPL {X  -159.990, Y  +620.788, Z    +0.000, E1   -23.368, E3 +464328.954}
SPL {X  -159.990, Y  +623.764, Z    +0.000, E1   -23.335, E3 +464343.646}
SPL {X  -159.990, Y  +625.941, Z    +0.000, E1   -23.337, E3 +464354.337}
SPL {X  -159.990, Y  +628.611, Z    +0.000, E1   -23.357, E3 +464367.416}
SPL {X  -159.990, Y  +631.169, Z    +0.000, E1   -23.338, E3 +464380.020}
SPL {X  -159.990, Y  +633.318, Z    +0.000, E1   -23.339, E3 +464390.610}
SPL {X  -159.990, Y  +635.650, Z    +0.000, E1   -23.339, E3 +464402.080}
SPL {X  -159.990, Y  +637.839, Z    +0.000, E1   -23.335, E3 +464412.891}
SPL {X  -159.990, Y  +640.072, Z    +0.000, E1   -23.325, E3 +464423.923}
SPL {X  -159.990, Y  +642.230, Z    +0.000, E1   -23.323, E3 +464434.605}
SPL {X  -159.990, Y  +645.287, Z    +0.000, E1   -23.340, E3 +464449.630}
SPL {X  -159.990, Y  +647.803, Z    +0.000, E1   -23.310, E3 +464462.107}
SPL {X  -159.990, Y  +650.790, Z    +0.000, E1   -23.346, E3 +464476.715}
SPL {X  -159.990, Y  +654.543, Z    +0.000, E1   -23.348, E3 +464495.168}
SPL {X  -159.990, Y  +658.319, Z    +0.000, E1   -23.349, E3 +464513.757}
SPL {X  -159.990, Y  +661.392, Z    +0.000, E1   -23.318, E3 +464528.960}
SPL {X  -159.990, Y  +663.662, Z    +0.000, E1   -23.322, E3 +464540.085}
SPL {X  -159.990, Y  +665.964, Z    +0.000, E1   -23.328, E3 +464551.375}
SPL {X  -159.990, Y  +667.870, Z    +0.000, E1   -23.320, E3 +464560.782}
SPL {X  -159.990, Y  +669.861, Z    +0.000, E1   -23.321, E3 +464570.583}
SPL {X  -159.983, Y  +672.946, Z    +0.000, E1   -23.359, E3 +464585.692}
SPL {X  -159.924, Y  +676.110, Z    +0.000, E1   -23.320, E3 +464601.391}
SPL {X  -159.845, Y  +678.302, Z    +0.000, E1   -23.298, E3 +464612.293}
SPL {X  -159.760, Y  +680.081, Z    +0.000, E1   -23.288, E3 +464621.137}
SPL {X  -159.626, Y  +682.287, Z    +0.000, E1   -23.280, E3 +464632.109}
SPL {X  -159.462, Y  +684.486, Z    +0.000, E1   -23.258, E3 +464643.108}
SPL {X  -159.246, Y  +686.911, Z    +0.000, E1   -23.230, E3 +464655.269}
SPL {X  -159.019, Y  +689.098, Z    +0.000, E1   -23.200, E3 +464666.271}
SPL {X  -158.660, Y  +692.086, Z    +0.000, E1   -23.176, E3 +464681.315}
ENDSPLINE

